LIN {X 0,Y 467.573,Z 511.242,A -85,B 0,C 180,E1 -7527.321,E2 -7527.321} C_VEL
LIN {X 0,Y 467.569,Z 511.24,A -85,B 0,C 180,E1 -7530.665,E2 -7530.665} C_VEL
LIN {X 0,Y 467.618,Z 511.239,A -85,B 0,C 180,E1 -7533.2,E2 -7533.2} C_VEL
LIN {X 0,Y 467.583,Z 511.237,A -85,B 0,C 180,E1 -7536.468,E2 -7536.468} C_VEL
LIN {X 0,Y 467.614,Z 511.233,A -85,B 0,C 180,E1 -7539.777,E2 -7539.777} C_VEL
LIN {X 0,Y 467.599,Z 511.235,A -85,B 0,C 180,E1 -7542.507,E2 -7542.507} C_VEL
LIN {X 0,Y 467.597,Z 511.242,A -85,B 0,C 180,E1 -7545.197,E2 -7545.197} C_VEL
LIN {X 0,Y 467.673,Z 511.225,A -85,B 0,C 180,E1 -7547.855,E2 -7547.855} C_VEL
LIN {X 0,Y 467.673,Z 511.231,A -85,B 0,C 180,E1 -7551.358,E2 -7551.358} C_VEL
LIN {X 0,Y 467.744,Z 511.216,A -85,B 0,C 180,E1 -7553.963,E2 -7553.963} C_VEL
LIN {X 0,Y 467.852,Z 511.208,A -85,B 0,C 180,E1 -7557.417,E2 -7557.417} C_VEL
LIN {X 0,Y 467.873,Z 511.2,A -85,B 0,C 180,E1 -7560,E2 -7560} C_VEL
LIN {X 0,Y 467.858,Z 511.203,A -85,B 0,C 180,E1 -7562.583,E2 -7562.583} C_VEL
LIN {X 0,Y 467.745,Z 511.216,A -85,B 0,C 180,E1 -7566.038,E2 -7566.038} C_VEL
LIN {X 0,Y 467.674,Z 511.226,A -85,B 0,C 180,E1 -7568.643,E2 -7568.643} C_VEL
LIN {X 0,Y 467.648,Z 511.228,A -85,B 0,C 180,E1 -7572.146,E2 -7572.146} C_VEL
LIN {X 0,Y 467.63,Z 511.233,A -85,B 0,C 180,E1 -7575.696,E2 -7575.696} C_VEL
LIN {X 0,Y 467.61,Z 511.235,A -85,B 0,C 180,E1 -7578.765,E2 -7578.765} C_VEL
LIN {X 0,Y 467.573,Z 511.246,A -85,B 0,C 180,E1 -7581.269,E2 -7581.269} C_VEL
LIN {X 0,Y 467.566,Z 511.239,A -85,B 0,C 180,E1 -7583.944,E2 -7583.944} C_VEL
LIN {X 0,Y 467.621,Z 511.233,A -85,B 0,C 180,E1 -7586.8,E2 -7586.8} C_VEL
LIN {X 0,Y 467.583,Z 511.239,A -85,B 0,C 180,E1 -7589.737,E2 -7589.737} C_VEL
LIN {X 0,Y 467.578,Z 511.238,A -85,B 0,C 180,E1 -7592.759,E2 -7592.759} C_VEL
LIN {X 0,Y 467.552,Z 511.241,A -85,B 0,C 180,E1 -7595.89,E2 -7595.89} C_VEL
LIN {X 0,Y 467.578,Z 511.242,A -85,B 0,C 180,E1 -7599.146,E2 -7599.146} C_VEL
LIN {X 0,Y 467.583,Z 511.236,A -85,B 0,C 180,E1 -7602.568,E2 -7602.568} C_VEL
LIN {X 0,Y 467.567,Z 511.242,A -85,B 0,C 180,E1 -7605.054,E2 -7605.054} C_VEL
LIN {X 0,Y 467.622,Z 511.238,A -85,B 0,C 180,E1 -7607.445,E2 -7607.445} C_VEL
LIN {X 0,Y 467.613,Z 511.234,A -85,B 0,C 180,E1 -7610.86,E2 -7610.86} C_VEL
LIN {X 0,Y 467.561,Z 511.239,A -85,B 0,C 180,E1 -7614.261,E2 -7614.261} C_VEL
LIN {X 0,Y 467.582,Z 511.244,A -85,B 0,C 180,E1 -7617.322,E2 -7617.322} C_VEL
LIN {X 0,Y 467.57,Z 511.242,A -85,B 0,C 180,E1 -7620.668,E2 -7620.668} C_VEL
LIN {X 0,Y 467.685,Z 511.313,A -85,B 0,C 180,E1 -7622.784,E2 -7622.784} C_VEL
LIN {X 0,Y 470.344,Z 524.929,A -85,B 0,C 180,E1 -7625.268,E2 -7625.268} C_VEL
LIN {X 0,Y 469.76,Z 538.705,A -85,B 0,C 180,E1 -7627.574,E2 -7627.574} C_VEL
LIN {X 0,Y 468.885,Z 558.208,A -85,B 0,C 180,E1 -7630.786,E2 -7630.786} C_VEL
LIN {X 0,Y 468.378,Z 571.672,A -85,B 0,C 180,E1 -7632.979,E2 -7632.979} C_VEL
LIN {X 0,Y 471.177,Z 592.338,A -85,B 0,C 180,E1 -7633.414,E2 -7633.414} C_VEL
LIN {X 0,Y 470.446,Z 679.842,A -85,B 0,C 180,E1 -7634.79,E2 -7634.79} C_VEL
LIN {X 0,Y 470.108,Z 692.551,A -85,B 0,C 180,E1 -7635.139,E2 -7635.139} C_VEL
LIN {X 0,Y 469.678,Z 705.019,A -85,B 0,C 180,E1 -7635.651,E2 -7635.651} C_VEL
LIN {X 0,Y 469.158,Z 717.567,A -85,B 0,C 180,E1 -7636.354,E2 -7636.354} C_VEL
LIN {X 0,Y 468.644,Z 729.795,A -85,B 0,C 180,E1 -7637.261,E2 -7637.261} C_VEL
LIN {X 0,Y 468.237,Z 739.902,A -85,B 0,C 180,E1 -7638.2,E2 -7638.2} C_VEL
LIN {X 0,Y 467.747,Z 748.542,A -85,B 0,C 180,E1 -7639.175,E2 -7639.175} C_VEL
LIN {X 0,Y 467.406,Z 756.518,A -85,B 0,C 180,E1 -7640.261,E2 -7640.261} C_VEL
LIN {X 0,Y 467.107,Z 764.316,A -85,B 0,C 180,E1 -7641.565,E2 -7641.565} C_VEL
LIN {X 0,Y 466.859,Z 771.486,A -85,B 0,C 180,E1 -7643.083,E2 -7643.083} C_VEL
LIN {X 0,Y 466.781,Z 776.263,A -85,B 0,C 180,E1 -7644.384,E2 -7644.384} C_VEL
LIN {X 0,Y 466.664,Z 779.908,A -85,B 0,C 180,E1 -7645.682,E2 -7645.682} C_VEL
LIN {X 0,Y 466.728,Z 781.794,A -85,B 0,C 180,E1 -7646.547,E2 -7646.547} C_VEL
LIN {X 0,Y 466.701,Z 783.202,A -85,B 0,C 180,E1 -7647.411,E2 -7647.411} C_VEL
LIN {X 0,Y 466.693,Z 784.204,A -85,B 0,C 180,E1 -7648.274,E2 -7648.274} C_VEL
LIN {X 0,Y 466.599,Z 785.018,A -85,B 0,C 180,E1 -7650,E2 -7650} C_VEL
LIN {X 0,Y 466.693,Z 784.171,A -85,B 0,C 180,E1 -7651.726,E2 -7651.726} C_VEL
LIN {X 0,Y 466.701,Z 783.153,A -85,B 0,C 180,E1 -7652.589,E2 -7652.589} C_VEL
LIN {X 0,Y 466.729,Z 781.728,A -85,B 0,C 180,E1 -7653.453,E2 -7653.453} C_VEL
LIN {X 0,Y 466.696,Z 778.735,A -85,B 0,C 180,E1 -7654.751,E2 -7654.751} C_VEL
LIN {X 0,Y 466.765,Z 774.695,A -85,B 0,C 180,E1 -7656.05,E2 -7656.05} C_VEL
LIN {X 0,Y 466.927,Z 768.484,A -85,B 0,C 180,E1 -7657.568,E2 -7657.568} C_VEL
LIN {X 0,Y 467.148,Z 761.707,A -85,B 0,C 180,E1 -7658.871,E2 -7658.871} C_VEL
LIN {X 0,Y 467.479,Z 753.307,A -85,B 0,C 180,E1 -7660.174,E2 -7660.174} C_VEL
LIN {X 0,Y 467.908,Z 744.688,A -85,B 0,C 180,E1 -7661.26,E2 -7661.26} C_VEL
LIN {X 0,Y 468.351,Z 734.541,A -85,B 0,C 180,E1 -7662.301,E2 -7662.301} C_VEL
LIN {X 0,Y 468.939,Z 723.534,A -85,B 0,C 180,E1 -7663.212,E2 -7663.212} C_VEL
LIN {X 0,Y 469.348,Z 711.968,A -85,B 0,C 180,E1 -7663.972,E2 -7663.972} C_VEL
LIN {X 0,Y 469.843,Z 698.703,A -85,B 0,C 180,E1 -7664.62,E2 -7664.62} C_VEL
LIN {X 0,Y 470.25,Z 685.293,A -85,B 0,C 180,E1 -7665.078,E2 -7665.078} C_VEL
LIN {X 0,Y 470.545,Z 671.932,A -85,B 0,C 180,E1 -7665.345,E2 -7665.345} C_VEL
LIN {X 0,Y 471.04,Z 590.105,A -85,B 0,C 180,E1 -7666.624,E2 -7666.624} C_VEL
LIN {X 0,Y 468.329,Z 570.989,A -85,B 0,C 180,E1 -7667.044,E2 -7667.044} C_VEL
LIN {X 0,Y 469.127,Z 550.502,A -85,B 0,C 180,E1 -7670.383,E2 -7670.383} C_VEL
LIN {X 0,Y 469.926,Z 532.596,A -85,B 0,C 180,E1 -7673.348,E2 -7673.348} C_VEL
LIN {X 0,Y 470.213,Z 524.341,A -85,B 0,C 180,E1 -7674.739,E2 -7674.739} C_VEL
LIN {X 0,Y 467.69,Z 511.23,A -85,B 0,C 180,E1 -7677.16,E2 -7677.16} C_VEL
LIN {X 0,Y 467.571,Z 511.246,A -85,B 0,C 180,E1 -7680.733,E2 -7680.733} C_VEL
LIN {X 0,Y 467.586,Z 511.241,A -85,B 0,C 180,E1 -7683.787,E2 -7683.787} C_VEL
LIN {X 0,Y 467.55,Z 511.244,A -85,B 0,C 180,E1 -7687.186,E2 -7687.186} C_VEL
LIN {X 0,Y 467.594,Z 511.239,A -85,B 0,C 180,E1 -7690.262,E2 -7690.262} C_VEL
LIN {X 0,Y 467.617,Z 511.239,A -85,B 0,C 180,E1 -7692.57,E2 -7692.57} C_VEL
LIN {X 0,Y 467.563,Z 511.241,A -85,B 0,C 180,E1 -7696.176,E2 -7696.176} C_VEL
LIN {X 0,Y 467.578,Z 511.244,A -85,B 0,C 180,E1 -7698.722,E2 -7698.722} C_VEL
LIN {X 0,Y 467.562,Z 511.24,A -85,B 0,C 180,E1 -7701.955,E2 -7701.955} C_VEL
LIN {X 0,Y 467.563,Z 511.241,A -85,B 0,C 180,E1 -7705.167,E2 -7705.167} C_VEL
LIN {X 0,Y 467.58,Z 511.239,A -85,B 0,C 180,E1 -7708.259,E2 -7708.259} C_VEL
LIN {X 0,Y 467.577,Z 511.239,A -85,B 0,C 180,E1 -7711.25,E2 -7711.25} C_VEL
LIN {X 0,Y 467.605,Z 511.235,A -85,B 0,C 180,E1 -7714.159,E2 -7714.159} C_VEL
LIN {X 0,Y 467.569,Z 511.245,A -85,B 0,C 180,E1 -7716.995,E2 -7716.995} C_VEL
LIN {X 0,Y 467.616,Z 511.231,A -85,B 0,C 180,E1 -7719.776,E2 -7719.776} C_VEL
LIN {X 0,Y 467.601,Z 511.237,A -85,B 0,C 180,E1 -7722.506,E2 -7722.506} C_VEL
LIN {X 0,Y 467.598,Z 511.238,A -85,B 0,C 180,E1 -7725.196,E2 -7725.196} C_VEL
LIN {X 0,Y 467.648,Z 511.229,A -85,B 0,C 180,E1 -7727.854,E2 -7727.854} C_VEL
LIN {X 0,Y 467.674,Z 511.229,A -85,B 0,C 180,E1 -7731.357,E2 -7731.357} C_VEL
LIN {X 0,Y 467.745,Z 511.214,A -85,B 0,C 180,E1 -7733.962,E2 -7733.962} C_VEL
LIN {X 0,Y 467.851,Z 511.206,A -85,B 0,C 180,E1 -7737.417,E2 -7737.417} C_VEL
LIN {X 0,Y 467.873,Z 511.199,A -85,B 0,C 180,E1 -7740,E2 -7740} C_VEL
LIN {X 0,Y 467.852,Z 511.206,A -85,B 0,C 180,E1 -7742.583,E2 -7742.583} C_VEL
LIN {X 0,Y 467.745,Z 511.216,A -85,B 0,C 180,E1 -7746.037,E2 -7746.037} C_VEL
LIN {X 0,Y 467.673,Z 511.229,A -85,B 0,C 180,E1 -7748.642,E2 -7748.642} C_VEL
LIN {X 0,Y 467.647,Z 511.229,A -85,B 0,C 180,E1 -7752.145,E2 -7752.145} C_VEL
LIN {X 0,Y 467.629,Z 511.233,A -85,B 0,C 180,E1 -7755.695,E2 -7755.695} C_VEL
LIN {X 0,Y 467.608,Z 511.238,A -85,B 0,C 180,E1 -7758.765,E2 -7758.765} C_VEL
LIN {X 0,Y 467.571,Z 511.246,A -85,B 0,C 180,E1 -7761.268,E2 -7761.268} C_VEL
LIN {X 0,Y 467.563,Z 511.244,A -85,B 0,C 180,E1 -7763.943,E2 -7763.943} C_VEL
LIN {X 0,Y 467.618,Z 511.241,A -85,B 0,C 180,E1 -7766.8,E2 -7766.8} C_VEL
LIN {X 0,Y 467.578,Z 511.243,A -85,B 0,C 180,E1 -7769.736,E2 -7769.736} C_VEL
LIN {X 0,Y 467.629,Z 511.278,A -85,B 0,C 180,E1 -7772.383,E2 -7772.383} C_VEL
LIN {X 0,Y 468.698,Z 518.116,A -85,B 0,C 180,E1 -7774.066,E2 -7774.066} C_VEL
LIN {X 0,Y 468.606,Z 522.269,A -85,B 0,C 180,E1 -7775.038,E2 -7775.038} C_VEL
LIN {X 0,Y 471.44,Z 535.638,A -85,B 0,C 180,E1 -7775.384,E2 -7775.384} C_VEL
LIN {X 0,Y 470.589,Z 628.803,A -85,B 0,C 180,E1 -7776.865,E2 -7776.865} C_VEL
LIN {X 0,Y 470.3,Z 642.7,A -85,B 0,C 180,E1 -7777.278,E2 -7777.278} C_VEL
LIN {X 0,Y 470.018,Z 654.766,A -85,B 0,C 180,E1 -7777.81,E2 -7777.81} C_VEL
LIN {X 0,Y 469.536,Z 666.953,A -85,B 0,C 180,E1 -7778.538,E2 -7778.538} C_VEL
LIN {X 0,Y 469.053,Z 678.321,A -85,B 0,C 180,E1 -7779.413,E2 -7779.413} C_VEL
LIN {X 0,Y 468.519,Z 688.987,A -85,B 0,C 180,E1 -7780.448,E2 -7780.448} C_VEL
LIN {X 0,Y 468.053,Z 698.759,A -85,B 0,C 180,E1 -7781.637,E2 -7781.637} C_VEL
LIN {X 0,Y 467.629,Z 706.828,A -85,B 0,C 180,E1 -7782.847,E2 -7782.847} C_VEL
LIN {X 0,Y 467.334,Z 713.616,A -85,B 0,C 180,E1 -7784.105,E2 -7784.105} C_VEL
LIN {X 0,Y 467.068,Z 719.943,A -85,B 0,C 180,E1 -7785.599,E2 -7785.599} C_VEL
LIN {X 0,Y 466.933,Z 723.941,A -85,B 0,C 180,E1 -7786.81,E2 -7786.81} C_VEL
LIN {X 0,Y 466.808,Z 727.024,A -85,B 0,C 180,E1 -7788.02,E2 -7788.02} C_VEL
LIN {X 0,Y 466.633,Z 729.788,A -85,B 0,C 180,E1 -7789.638,E2 -7789.638} C_VEL
LIN {X 0,Y 466.57,Z 730.886,A -85,B 0,C 180,E1 -7790.755,E2 -7790.755} C_VEL
LIN {X 0,Y 466.575,Z 731.291,A -85,B 0,C 180,E1 -7791.861,E2 -7791.861} C_VEL
LIN {X 0,Y 466.571,Z 731.055,A -85,B 0,C 180,E1 -7792.971,E2 -7792.971} C_VEL
LIN {X 0,Y 466.6,Z 729.522,A -85,B 0,C 180,E1 -7794.588,E2 -7794.588} C_VEL
LIN {X 0,Y 466.766,Z 726.76,A -85,B 0,C 180,E1 -7796.145,E2 -7796.145} C_VEL
LIN {X 0,Y 466.914,Z 723.325,A -85,B 0,C 180,E1 -7797.448,E2 -7797.448} C_VEL
LIN {X 0,Y 466.999,Z 720.883,A -85,B 0,C 180,E1 -7798.19,E2 -7798.19} C_VEL
LIN {X 0,Y 466.47,Z 718.546,A -85,B 0,C 180,E1 -7798.854,E2 -7798.854} C_VEL
LIN {X 0,Y 463.785,Z 714.337,A -85,B 0,C 180,E1 -7799.912,E2 -7799.912} C_VEL
LIN {X 0,Y 461.138,Z 709.44,A -85,B 0,C 180,E1 -7800.934,E2 -7800.934} C_VEL
LIN {X 0,Y 460.675,Z 706.022,A -85,B 0,C 180,E1 -7801.532,E2 -7801.532} C_VEL
LIN {X 0,Y 461.128,Z 697.482,A -85,B 0,C 180,E1 -7802.792,E2 -7802.792} C_VEL
LIN {X 0,Y 461.645,Z 688.03,A -85,B 0,C 180,E1 -7803.922,E2 -7803.922} C_VEL
LIN {X 0,Y 462.119,Z 677.677,A -85,B 0,C 180,E1 -7804.918,E2 -7804.918} C_VEL
LIN {X 0,Y 462.601,Z 666.443,A -85,B 0,C 180,E1 -7805.784,E2 -7805.784} C_VEL
LIN {X 0,Y 463.087,Z 653.998,A -85,B 0,C 180,E1 -7806.524,E2 -7806.524} C_VEL
LIN {X 0,Y 463.455,Z 640.905,A -85,B 0,C 180,E1 -7807.088,E2 -7807.088} C_VEL
LIN {X 0,Y 463.693,Z 627.903,A -85,B 0,C 180,E1 -7807.463,E2 -7807.463} C_VEL
LIN {X 0,Y 464.487,Z 535.776,A -85,B 0,C 180,E1 -7808.94,E2 -7808.94} C_VEL
LIN {X 0,Y 461.511,Z 521.937,A -85,B 0,C 180,E1 -7809.294,E2 -7809.294} C_VEL
LIN {X 0,Y 461.424,Z 517.113,A -85,B 0,C 180,E1 -7810.423,E2 -7810.423} C_VEL
LIN {X 0,Y 460.618,Z 512.11,A -85,B 0,C 180,E1 -7811.658,E2 -7811.658} C_VEL
LIN {X 0,Y 460.562,Z 512.118,A -85,B 0,C 180,E1 -7814.965,E2 -7814.965} C_VEL
LIN {X 0,Y 460.608,Z 512.109,A -85,B 0,C 180,E1 -7818.559,E2 -7818.559} C_VEL
LIN {X 0,Y 460.692,Z 512.095,A -85,B 0,C 180,E1 -7822.109,E2 -7822.109} C_VEL
LIN {X 0,Y 460.692,Z 512.101,A -85,B 0,C 180,E1 -7824.748,E2 -7824.748} C_VEL
LIN {X 0,Y 460.823,Z 512.08,A -85,B 0,C 180,E1 -7827.378,E2 -7827.378} C_VEL
LIN {X 0,Y 460.851,Z 512.075,A -85,B 0,C 180,E1 -7830,E2 -7830} C_VEL
LIN {X 0,Y 460.822,Z 512.082,A -85,B 0,C 180,E1 -7832.622,E2 -7832.622} C_VEL
LIN {X 0,Y 460.709,Z 512.093,A -85,B 0,C 180,E1 -7836.13,E2 -7836.13} C_VEL
LIN {X 0,Y 460.626,Z 512.109,A -85,B 0,C 180,E1 -7838.776,E2 -7838.776} C_VEL
LIN {X 0,Y 460.61,Z 512.107,A -85,B 0,C 180,E1 -7842.445,E2 -7842.445} C_VEL
LIN {X 0,Y 460.596,Z 512.106,A -85,B 0,C 180,E1 -7845.997,E2 -7845.997} C_VEL
LIN {X 0,Y 460.567,Z 512.117,A -85,B 0,C 180,E1 -7848.902,E2 -7848.902} C_VEL
LIN {X 0,Y 460.512,Z 512.119,A -85,B 0,C 180,E1 -7851.485,E2 -7851.485} C_VEL
LIN {X 0,Y 460.538,Z 512.114,A -85,B 0,C 180,E1 -7854.332,E2 -7854.332} C_VEL
LIN {X 0,Y 460.575,Z 512.114,A -85,B 0,C 180,E1 -7857.243,E2 -7857.243} C_VEL
LIN {X 0,Y 460.526,Z 512.115,A -85,B 0,C 180,E1 -7860.238,E2 -7860.238} C_VEL
LIN {X 0,Y 460.523,Z 512.12,A -85,B 0,C 180,E1 -7863.324,E2 -7863.324} C_VEL
LIN {X 0,Y 460.474,Z 512.124,A -85,B 0,C 180,E1 -7866.529,E2 -7866.529} C_VEL
LIN {X 0,Y 460.572,Z 512.109,A -85,B 0,C 180,E1 -7869.857,E2 -7869.857} C_VEL
LIN {X 0,Y 460.536,Z 512.12,A -85,B 0,C 180,E1 -7872.904,E2 -7872.904} C_VEL
LIN {X 0,Y 460.516,Z 512.117,A -85,B 0,C 180,E1 -7875.828,E2 -7875.828} C_VEL
LIN {X 0,Y 460.535,Z 512.121,A -85,B 0,C 180,E1 -7878.99,E2 -7878.99} C_VEL
LIN {X 0,Y 460.539,Z 512.119,A -85,B 0,C 180,E1 -7881.269,E2 -7881.269} C_VEL
LIN {X 0,Y 460.505,Z 512.119,A -85,B 0,C 180,E1 -7884.555,E2 -7884.555} C_VEL
LIN {X 0,Y 460.523,Z 512.117,A -85,B 0,C 180,E1 -7887.716,E2 -7887.716} C_VEL
LIN {X 0,Y 460.538,Z 512.117,A -85,B 0,C 180,E1 -7890.769,E2 -7890.769} C_VEL
LIN {X 0,Y 460.559,Z 512.112,A -85,B 0,C 180,E1 -7893.735,E2 -7893.735} C_VEL
LIN {X 0,Y 460.536,Z 512.116,A -85,B 0,C 180,E1 -7896.624,E2 -7896.624} C_VEL
LIN {X 0,Y 460.542,Z 512.117,A -85,B 0,C 180,E1 -7899.453,E2 -7899.453} C_VEL
LIN {X 0,Y 460.549,Z 512.112,A -85,B 0,C 180,E1 -7902.23,E2 -7902.23} C_VEL
LIN {X 0,Y 460.555,Z 512.117,A -85,B 0,C 180,E1 -7904.965,E2 -7904.965} C_VEL
LIN {X 0,Y 460.62,Z 512.105,A -85,B 0,C 180,E1 -7907.667,E2 -7907.667} C_VEL
LIN {X 0,Y 460.62,Z 512.111,A -85,B 0,C 180,E1 -7911.224,E2 -7911.224} C_VEL
LIN {X 0,Y 460.709,Z 512.093,A -85,B 0,C 180,E1 -7913.871,E2 -7913.871} C_VEL
LIN {X 0,Y 460.817,Z 512.085,A -85,B 0,C 180,E1 -7917.378,E2 -7917.378} C_VEL
LIN {X 0,Y 460.844,Z 512.076,A -85,B 0,C 180,E1 -7920,E2 -7920} C_VEL
LIN {X 0,Y 460.824,Z 512.079,A -85,B 0,C 180,E1 -7922.623,E2 -7922.623} C_VEL
LIN {X 0,Y 460.71,Z 512.092,A -85,B 0,C 180,E1 -7926.13,E2 -7926.13} C_VEL
LIN {X 0,Y 460.621,Z 512.106,A -85,B 0,C 180,E1 -7928.777,E2 -7928.777} C_VEL
LIN {X 0,Y 460.604,Z 512.106,A -85,B 0,C 180,E1 -7932.446,E2 -7932.446} C_VEL
LIN {X 0,Y 460.592,Z 512.107,A -85,B 0,C 180,E1 -7935.998,E2 -7935.998} C_VEL
LIN {X 0,Y 460.563,Z 512.114,A -85,B 0,C 180,E1 -7938.903,E2 -7938.903} C_VEL
LIN {X 0,Y 460.508,Z 512.123,A -85,B 0,C 180,E1 -7941.486,E2 -7941.486} C_VEL
LIN {X 0,Y 460.535,Z 512.114,A -85,B 0,C 180,E1 -7944.333,E2 -7944.333} C_VEL
LIN {X 0,Y 460.578,Z 512.116,A -85,B 0,C 180,E1 -7947.244,E2 -7947.244} C_VEL
LIN {X 0,Y 460.525,Z 512.115,A -85,B 0,C 180,E1 -7950.239,E2 -7950.239} C_VEL
LIN {X 0,Y 460.524,Z 512.124,A -85,B 0,C 180,E1 -7953.326,E2 -7953.326} C_VEL
LIN {X 0,Y 460.475,Z 512.122,A -85,B 0,C 180,E1 -7956.53,E2 -7956.53} C_VEL
LIN {X 0,Y 460.554,Z 512.113,A -85,B 0,C 180,E1 -7959.861,E2 -7959.861} C_VEL
LIN {X 0,Y 460.513,Z 512.119,A -85,B 0,C 180,E1 -7962.902,E2 -7962.902} C_VEL
LIN {X 0,Y 460.521,Z 512.118,A -85,B 0,C 180,E1 -7965.83,E2 -7965.83} C_VEL
LIN {X 0,Y 460.541,Z 512.117,A -85,B 0,C 180,E1 -7968.991,E2 -7968.991} C_VEL
LIN {X 0,Y 460.542,Z 512.12,A -85,B 0,C 180,E1 -7971.27,E2 -7971.27} C_VEL
LIN {X 0,Y 460.512,Z 512.117,A -85,B 0,C 180,E1 -7974.555,E2 -7974.555} C_VEL
LIN {X 0,Y 460.532,Z 512.121,A -85,B 0,C 180,E1 -7977.717,E2 -7977.717} C_VEL
LIN {X 0,Y 460.54,Z 512.118,A -85,B 0,C 180,E1 -7980.77,E2 -7980.77} C_VEL
LIN {X 0,Y 460.637,Z 512.174,A -85,B 0,C 180,E1 -7982.554,E2 -7982.554} C_VEL
LIN {X 0,Y 463.311,Z 525.627,A -85,B 0,C 180,E1 -7985.055,E2 -7985.055} C_VEL
LIN {X 0,Y 463.231,Z 531.441,A -85,B 0,C 180,E1 -7986.057,E2 -7986.057} C_VEL
LIN {X 0,Y 462.345,Z 549.328,A -85,B 0,C 180,E1 -7989.071,E2 -7989.071} C_VEL
LIN {X 0,Y 461.463,Z 569.802,A -85,B 0,C 180,E1 -7992.473,E2 -7992.473} C_VEL
LIN {X 0,Y 461.394,Z 571.264,A -85,B 0,C 180,E1 -7992.713,E2 -7992.713} C_VEL
LIN {X 0,Y 464.355,Z 592.628,A -85,B 0,C 180,E1 -7993.179,E2 -7993.179} C_VEL
LIN {X 0,Y 463.544,Z 680.366,A -85,B 0,C 180,E1 -7994.586,E2 -7994.586} C_VEL
LIN {X 0,Y 463.158,Z 693.499,A -85,B 0,C 180,E1 -7994.967,E2 -7994.967} C_VEL
LIN {X 0,Y 462.688,Z 706.737,A -85,B 0,C 180,E1 -7995.542,E2 -7995.542} C_VEL
LIN {X 0,Y 462.156,Z 718.676,A -85,B 0,C 180,E1 -7996.255,E2 -7996.255} C_VEL
LIN {X 0,Y 461.625,Z 730.429,A -85,B 0,C 180,E1 -7997.159,E2 -7997.159} C_VEL
LIN {X 0,Y 461.203,Z 740.514,A -85,B 0,C 180,E1 -7998.129,E2 -7998.129} C_VEL
LIN {X 0,Y 460.633,Z 749.81,A -85,B 0,C 180,E1 -7999.228,E2 -7999.228} C_VEL
LIN {X 0,Y 460.215,Z 758.854,A -85,B 0,C 180,E1 -8000.552,E2 -8000.552} C_VEL
LIN {X 0,Y 459.936,Z 766.143,A -85,B 0,C 180,E1 -8001.875,E2 -8001.875} C_VEL
LIN {X 0,Y 459.747,Z 772.252,A -85,B 0,C 180,E1 -8003.273,E2 -8003.273} C_VEL
LIN {X 0,Y 459.679,Z 777.178,A -85,B 0,C 180,E1 -8004.737,E2 -8004.737} C_VEL
LIN {X 0,Y 459.579,Z 779.494,A -85,B 0,C 180,E1 -8005.615,E2 -8005.615} C_VEL
LIN {X 0,Y 459.626,Z 781.382,A -85,B 0,C 180,E1 -8006.494,E2 -8006.494} C_VEL
LIN {X 0,Y 459.621,Z 782.794,A -85,B 0,C 180,E1 -8007.371,E2 -8007.371} C_VEL
LIN {X 0,Y 459.63,Z 783.797,A -85,B 0,C 180,E1 -8008.248,E2 -8008.248} C_VEL
LIN {X 0,Y 459.531,Z 784.611,A -85,B 0,C 180,E1 -8010,E2 -8010} C_VEL
LIN {X 0,Y 459.63,Z 783.763,A -85,B 0,C 180,E1 -8011.752,E2 -8011.752} C_VEL
LIN {X 0,Y 459.621,Z 782.742,A -85,B 0,C 180,E1 -8012.629,E2 -8012.629} C_VEL
LIN {X 0,Y 459.626,Z 781.315,A -85,B 0,C 180,E1 -8013.506,E2 -8013.506} C_VEL
LIN {X 0,Y 459.627,Z 778.32,A -85,B 0,C 180,E1 -8014.824,E2 -8014.824} C_VEL
LIN {X 0,Y 459.715,Z 773.225,A -85,B 0,C 180,E1 -8016.431,E2 -8016.431} C_VEL
LIN {X 0,Y 459.891,Z 767.031,A -85,B 0,C 180,E1 -8017.905,E2 -8017.905} C_VEL
LIN {X 0,Y 460.181,Z 760.022,A -85,B 0,C 180,E1 -8019.227,E2 -8019.227} C_VEL
LIN {X 0,Y 460.532,Z 751.247,A -85,B 0,C 180,E1 -8020.552,E2 -8020.552} C_VEL
LIN {X 0,Y 461.034,Z 742.268,A -85,B 0,C 180,E1 -8021.653,E2 -8021.653} C_VEL
LIN {X 0,Y 461.56,Z 731.528,A -85,B 0,C 180,E1 -8022.726,E2 -8022.726} C_VEL
LIN {X 0,Y 462.095,Z 720.024,A -85,B 0,C 180,E1 -8023.635,E2 -8023.635} C_VEL
LIN {X 0,Y 462.63,Z 707.504,A -85,B 0,C 180,E1 -8024.404,E2 -8024.404} C_VEL
LIN {X 0,Y 463.15,Z 694.847,A -85,B 0,C 180,E1 -8024.977,E2 -8024.977} C_VEL
LIN {X 0,Y 463.495,Z 682.598,A -85,B 0,C 180,E1 -8025.359,E2 -8025.359} C_VEL
LIN {X 0,Y 463.857,Z 662.673,A -85,B 0,C 180,E1 -8025.713,E2 -8025.713} C_VEL
LIN {X 0,Y 464.27,Z 591.113,A -85,B 0,C 180,E1 -8026.856,E2 -8026.856} C_VEL
LIN {X 0,Y 461.349,Z 570.475,A -85,B 0,C 180,E1 -8027.326,E2 -8027.326} C_VEL
LIN {X 0,Y 462.145,Z 551.497,A -85,B 0,C 180,E1 -8030.473,E2 -8030.473} C_VEL
LIN {X 0,Y 463.065,Z 532.253,A -85,B 0,C 180,E1 -8033.715,E2 -8033.715} C_VEL
LIN {X 0,Y 463.211,Z 525.142,A -85,B 0,C 180,E1 -8034.942,E2 -8034.942} C_VEL
LIN {X 0,Y 460.617,Z 512.11,A -85,B 0,C 180,E1 -8037.406,E2 -8037.406} C_VEL
LIN {X 0,Y 460.511,Z 512.124,A -85,B 0,C 180,E1 -8040.239,E2 -8040.239} C_VEL
LIN {X 0,Y 460.529,Z 512.121,A -85,B 0,C 180,E1 -8043.324,E2 -8043.324} C_VEL
LIN {X 0,Y 460.478,Z 512.13,A -85,B 0,C 180,E1 -8046.528,E2 -8046.528} C_VEL
LIN {X 0,Y 460.574,Z 512.111,A -85,B 0,C 180,E1 -8049.857,E2 -8049.857} C_VEL
LIN {X 0,Y 460.54,Z 512.119,A -85,B 0,C 180,E1 -8052.903,E2 -8052.903} C_VEL
LIN {X 0,Y 460.516,Z 512.117,A -85,B 0,C 180,E1 -8055.828,E2 -8055.828} C_VEL
LIN {X 0,Y 460.53,Z 512.12,A -85,B 0,C 180,E1 -8058.988,E2 -8058.988} C_VEL
LIN {X 0,Y 460.522,Z 512.119,A -85,B 0,C 180,E1 -8061.266,E2 -8061.266} C_VEL
LIN {X 0,Y 460.509,Z 512.123,A -85,B 0,C 180,E1 -8064.554,E2 -8064.554} C_VEL
LIN {X 0,Y 460.527,Z 512.116,A -85,B 0,C 180,E1 -8067.715,E2 -8067.715} C_VEL
LIN {X 0,Y 460.541,Z 512.121,A -85,B 0,C 180,E1 -8070.769,E2 -8070.769} C_VEL
LIN {X 0,Y 460.561,Z 512.112,A -85,B 0,C 180,E1 -8073.734,E2 -8073.734} C_VEL
LIN {X 0,Y 460.539,Z 512.116,A -85,B 0,C 180,E1 -8076.623,E2 -8076.623} C_VEL
LIN {X 0,Y 460.544,Z 512.114,A -85,B 0,C 180,E1 -8079.452,E2 -8079.452} C_VEL
LIN {X 0,Y 460.551,Z 512.113,A -85,B 0,C 180,E1 -8082.229,E2 -8082.229} C_VEL
LIN {X 0,Y 460.557,Z 512.119,A -85,B 0,C 180,E1 -8084.964,E2 -8084.964} C_VEL
LIN {X 0,Y 460.601,Z 512.107,A -85,B 0,C 180,E1 -8087.665,E2 -8087.665} C_VEL
LIN {X 0,Y 460.621,Z 512.109,A -85,B 0,C 180,E1 -8091.223,E2 -8091.223} C_VEL
LIN {X 0,Y 460.709,Z 512.09,A -85,B 0,C 180,E1 -8093.87,E2 -8093.87} C_VEL
LIN {X 0,Y 460.817,Z 512.082,A -85,B 0,C 180,E1 -8097.377,E2 -8097.377} C_VEL
LIN {X 0,Y 460.844,Z 512.075,A -85,B 0,C 180,E1 -8100,E2 -8100} C_VEL
LIN {X 0,Y 460.817,Z 512.083,A -85,B 0,C 180,E1 -8102.622,E2 -8102.622} C_VEL
LIN {X 0,Y 460.709,Z 512.092,A -85,B 0,C 180,E1 -8106.129,E2 -8106.129} C_VEL
LIN {X 0,Y 460.62,Z 512.109,A -85,B 0,C 180,E1 -8108.776,E2 -8108.776} C_VEL
LIN {X 0,Y 460.603,Z 512.108,A -85,B 0,C 180,E1 -8112.445,E2 -8112.445} C_VEL
LIN {X 0,Y 460.59,Z 512.109,A -85,B 0,C 180,E1 -8115.997,E2 -8115.997} C_VEL
LIN {X 0,Y 460.561,Z 512.118,A -85,B 0,C 180,E1 -8118.902,E2 -8118.902} C_VEL
LIN {X 0,Y 460.506,Z 512.124,A -85,B 0,C 180,E1 -8121.486,E2 -8121.486} C_VEL
LIN {X 0,Y 460.533,Z 512.12,A -85,B 0,C 180,E1 -8124.332,E2 -8124.332} C_VEL
LIN {X 0,Y 460.574,Z 512.119,A -85,B 0,C 180,E1 -8127.243,E2 -8127.243} C_VEL
LIN {X 0,Y 460.518,Z 512.121,A -85,B 0,C 180,E1 -8130.239,E2 -8130.239} C_VEL
LIN {X 0,Y 460.613,Z 512.276,A -85,B 0,C 180,E1 -8132.213,E2 -8132.213} C_VEL
LIN {X 0,Y 461.745,Z 519.491,A -85,B 0,C 180,E1 -8134.011,E2 -8134.011} C_VEL
LIN {X 0,Y 461.686,Z 522.905,A -85,B 0,C 180,E1 -8134.793,E2 -8134.793} C_VEL
LIN {X 0,Y 464.681,Z 536.46,A -85,B 0,C 180,E1 -8135.136,E2 -8135.136} C_VEL
LIN {X 0,Y 463.762,Z 629.077,A -85,B 0,C 180,E1 -8136.631,E2 -8136.631} C_VEL
LIN {X 0,Y 463.473,Z 642.341,A -85,B 0,C 180,E1 -8137.025,E2 -8137.025} C_VEL
LIN {X 0,Y 463.188,Z 654.654,A -85,B 0,C 180,E1 -8137.568,E2 -8137.568} C_VEL
LIN {X 0,Y 462.718,Z 666.186,A -85,B 0,C 180,E1 -8138.251,E2 -8138.251} C_VEL
LIN {X 0,Y 462.195,Z 677.921,A -85,B 0,C 180,E1 -8139.152,E2 -8139.152} C_VEL
LIN {X 0,Y 461.723,Z 687.432,A -85,B 0,C 180,E1 -8140.062,E2 -8140.062} C_VEL
LIN {X 0,Y 461.2,Z 696.472,A -85,B 0,C 180,E1 -8141.115,E2 -8141.115} C_VEL
LIN {X 0,Y 460.73,Z 705.187,A -85,B 0,C 180,E1 -8142.37,E2 -8142.37} C_VEL
LIN {X 0,Y 460.376,Z 712.937,A -85,B 0,C 180,E1 -8143.764,E2 -8143.764} C_VEL
LIN {X 0,Y 460.094,Z 718.436,A -85,B 0,C 180,E1 -8144.997,E2 -8144.997} C_VEL
LIN {X 0,Y 459.889,Z 723.865,A -85,B 0,C 180,E1 -8146.554,E2 -8146.554} C_VEL
LIN {X 0,Y 459.783,Z 726.943,A -85,B 0,C 180,E1 -8147.736,E2 -8147.736} C_VEL
LIN {X 0,Y 459.604,Z 729.178,A -85,B 0,C 180,E1 -8148.889,E2 -8148.889} C_VEL
LIN {X 0,Y 459.515,Z 730.708,A -85,B 0,C 180,E1 -8150.033,E2 -8150.033} C_VEL
LIN {X 0,Y 459.482,Z 731.576,A -85,B 0,C 180,E1 -8151.266,E2 -8151.266} C_VEL
LIN {X 0,Y 459.473,Z 731.604,A -85,B 0,C 180,E1 -8152.69,E2 -8152.69} C_VEL
LIN {X 0,Y 459.516,Z 730.548,A -85,B 0,C 180,E1 -8154.154,E2 -8154.154} C_VEL
LIN {X 0,Y 459.622,Z 728.276,A -85,B 0,C 180,E1 -8155.659,E2 -8155.659} C_VEL
LIN {X 0,Y 459.846,Z 724.642,A -85,B 0,C 180,E1 -8157.201,E2 -8157.201} C_VEL
LIN {X 0,Y 460.048,Z 719.338,A -85,B 0,C 180,E1 -8158.813,E2 -8158.813} C_VEL
LIN {X 0,Y 460.308,Z 713.599,A -85,B 0,C 180,E1 -8160.143,E2 -8160.143} C_VEL
LIN {X 0,Y 460.675,Z 706.022,A -85,B 0,C 180,E1 -8161.532,E2 -8161.532} C_VEL
LIN {X 0,Y 460.136,Z 703.69,A -85,B 0,C 180,E1 -8161.927,E2 -8161.927} C_VEL
LIN {X 0,Y 454.869,Z 696.121,A -85,B 0,C 180,E1 -8163.166,E2 -8163.166} C_VEL
LIN {X 0,Y 454.431,Z 693.359,A -85,B 0,C 180,E1 -8163.529,E2 -8163.529} C_VEL
LIN {X 0,Y 454.925,Z 683.4,A -85,B 0,C 180,E1 -8164.616,E2 -8164.616} C_VEL
LIN {X 0,Y 455.496,Z 672.72,A -85,B 0,C 180,E1 -8165.55,E2 -8165.55} C_VEL
LIN {X 0,Y 456.001,Z 660.791,A -85,B 0,C 180,E1 -8166.378,E2 -8166.378} C_VEL
LIN {X 0,Y 456.421,Z 648.899,A -85,B 0,C 180,E1 -8167.001,E2 -8167.001} C_VEL
LIN {X 0,Y 456.739,Z 636.3,A -85,B 0,C 180,E1 -8167.475,E2 -8167.475} C_VEL
LIN {X 0,Y 456.979,Z 623.65,A -85,B 0,C 180,E1 -8167.776,E2 -8167.776} C_VEL
LIN {X 0,Y 457.757,Z 537.021,A -85,B 0,C 180,E1 -8169.175,E2 -8169.175} C_VEL
LIN {X 0,Y 454.588,Z 522.315,A -85,B 0,C 180,E1 -8169.556,E2 -8169.556} C_VEL
LIN {X 0,Y 454.375,Z 517.725,A -85,B 0,C 180,E1 -8170.648,E2 -8170.648} C_VEL
LIN {X 0,Y 453.565,Z 512.989,A -85,B 0,C 180,E1 -8171.83,E2 -8171.83} C_VEL
LIN {X 0,Y 453.537,Z 512.994,A -85,B 0,C 180,E1 -8174.727,E2 -8174.727} C_VEL
LIN {X 0,Y 453.557,Z 512.985,A -85,B 0,C 180,E1 -8178.379,E2 -8178.379} C_VEL
LIN {X 0,Y 453.649,Z 512.972,A -85,B 0,C 180,E1 -8181.985,E2 -8181.985} C_VEL
LIN {X 0,Y 453.665,Z 512.975,A -85,B 0,C 180,E1 -8184.667,E2 -8184.667} C_VEL
LIN {X 0,Y 453.763,Z 512.96,A -85,B 0,C 180,E1 -8187.337,E2 -8187.337} C_VEL
LIN {X 0,Y 453.821,Z 512.95,A -85,B 0,C 180,E1 -8190,E2 -8190} C_VEL
LIN {X 0,Y 453.763,Z 512.962,A -85,B 0,C 180,E1 -8192.663,E2 -8192.663} C_VEL
LIN {X 0,Y 453.676,Z 512.969,A -85,B 0,C 180,E1 -8196.225,E2 -8196.225} C_VEL
LIN {X 0,Y 453.589,Z 512.987,A -85,B 0,C 180,E1 -8198.913,E2 -8198.913} C_VEL
LIN {X 0,Y 453.56,Z 512.986,A -85,B 0,C 180,E1 -8202.529,E2 -8202.529} C_VEL
LIN {X 0,Y 453.541,Z 512.986,A -85,B 0,C 180,E1 -8206.196,E2 -8206.196} C_VEL
LIN {X 0,Y 453.517,Z 512.996,A -85,B 0,C 180,E1 -8209.041,E2 -8209.041} C_VEL
LIN {X 0,Y 453.472,Z 512.994,A -85,B 0,C 180,E1 -8211.836,E2 -8211.836} C_VEL
LIN {X 0,Y 453.51,Z 512.994,A -85,B 0,C 180,E1 -8214.734,E2 -8214.734} C_VEL
LIN {X 0,Y 453.534,Z 512.986,A -85,B 0,C 180,E1 -8217.961,E2 -8217.961} C_VEL
LIN {X 0,Y 453.479,Z 512.998,A -85,B 0,C 180,E1 -8220.758,E2 -8220.758} C_VEL
LIN {X 0,Y 453.472,Z 512.994,A -85,B 0,C 180,E1 -8223.912,E2 -8223.912} C_VEL
LIN {X 0,Y 453.466,Z 513.001,A -85,B 0,C 180,E1 -8227.187,E2 -8227.187} C_VEL
LIN {X 0,Y 453.527,Z 512.99,A -85,B 0,C 180,E1 -8229.445,E2 -8229.445} C_VEL
LIN {X 0,Y 453.485,Z 513,A -85,B 0,C 180,E1 -8232.991,E2 -8232.991} C_VEL
LIN {X 0,Y 453.469,Z 512.995,A -85,B 0,C 180,E1 -8235.78,E2 -8235.78} C_VEL
LIN {X 0,Y 453.488,Z 512.992,A -85,B 0,C 180,E1 -8238.211,E2 -8238.211} C_VEL
LIN {X 0,Y 453.524,Z 512.992,A -85,B 0,C 180,E1 -8240.787,E2 -8240.787} C_VEL
LIN {X 0,Y 453.449,Z 512.997,A -85,B 0,C 180,E1 -8243.917,E2 -8243.917} C_VEL
LIN {X 0,Y 453.474,Z 513.001,A -85,B 0,C 180,E1 -8247.151,E2 -8247.151} C_VEL
LIN {X 0,Y 453.505,Z 512.99,A -85,B 0,C 180,E1 -8250.271,E2 -8250.271} C_VEL
LIN {X 0,Y 453.504,Z 512.996,A -85,B 0,C 180,E1 -8253.294,E2 -8253.294} C_VEL
LIN {X 0,Y 453.494,Z 512.991,A -85,B 0,C 180,E1 -8256.239,E2 -8256.239} C_VEL
LIN {X 0,Y 453.474,Z 513.002,A -85,B 0,C 180,E1 -8259.118,E2 -8259.118} C_VEL
LIN {X 0,Y 453.502,Z 512.99,A -85,B 0,C 180,E1 -8261.945,E2 -8261.945} C_VEL
LIN {X 0,Y 453.53,Z 512.989,A -85,B 0,C 180,E1 -8264.726,E2 -8264.726} C_VEL
LIN {X 0,Y 453.592,Z 512.983,A -85,B 0,C 180,E1 -8267.472,E2 -8267.472} C_VEL
LIN {X 0,Y 453.584,Z 512.987,A -85,B 0,C 180,E1 -8271.087,E2 -8271.087} C_VEL
LIN {X 0,Y 453.675,Z 512.97,A -85,B 0,C 180,E1 -8273.775,E2 -8273.775} C_VEL
LIN {X 0,Y 453.758,Z 512.965,A -85,B 0,C 180,E1 -8277.337,E2 -8277.337} C_VEL
LIN {X 0,Y 453.814,Z 512.951,A -85,B 0,C 180,E1 -8280,E2 -8280} C_VEL
LIN {X 0,Y 453.765,Z 512.959,A -85,B 0,C 180,E1 -8282.664,E2 -8282.664} C_VEL
LIN {X 0,Y 453.676,Z 512.968,A -85,B 0,C 180,E1 -8286.226,E2 -8286.226} C_VEL
LIN {X 0,Y 453.585,Z 512.984,A -85,B 0,C 180,E1 -8288.914,E2 -8288.914} C_VEL
LIN {X 0,Y 453.555,Z 512.984,A -85,B 0,C 180,E1 -8292.53,E2 -8292.53} C_VEL
LIN {X 0,Y 453.537,Z 512.986,A -85,B 0,C 180,E1 -8296.197,E2 -8296.197} C_VEL
LIN {X 0,Y 453.513,Z 512.994,A -85,B 0,C 180,E1 -8299.042,E2 -8299.042} C_VEL
LIN {X 0,Y 453.469,Z 512.996,A -85,B 0,C 180,E1 -8301.837,E2 -8301.837} C_VEL
LIN {X 0,Y 453.507,Z 512.991,A -85,B 0,C 180,E1 -8304.735,E2 -8304.735} C_VEL
LIN {X 0,Y 453.532,Z 512.987,A -85,B 0,C 180,E1 -8307.962,E2 -8307.962} C_VEL
LIN {X 0,Y 453.479,Z 512.995,A -85,B 0,C 180,E1 -8310.76,E2 -8310.76} C_VEL
LIN {X 0,Y 453.473,Z 512.995,A -85,B 0,C 180,E1 -8313.914,E2 -8313.914} C_VEL
LIN {X 0,Y 453.466,Z 513.001,A -85,B 0,C 180,E1 -8317.189,E2 -8317.189} C_VEL
LIN {X 0,Y 453.513,Z 512.995,A -85,B 0,C 180,E1 -8319.448,E2 -8319.448} C_VEL
LIN {X 0,Y 453.465,Z 512.998,A -85,B 0,C 180,E1 -8322.995,E2 -8322.995} C_VEL
LIN {X 0,Y 453.474,Z 512.996,A -85,B 0,C 180,E1 -8325.781,E2 -8325.781} C_VEL
LIN {X 0,Y 453.494,Z 512.991,A -85,B 0,C 180,E1 -8328.212,E2 -8328.212} C_VEL
LIN {X 0,Y 453.529,Z 512.988,A -85,B 0,C 180,E1 -8330.789,E2 -8330.789} C_VEL
LIN {X 0,Y 453.455,Z 512.998,A -85,B 0,C 180,E1 -8333.918,E2 -8333.918} C_VEL
LIN {X 0,Y 453.483,Z 513,A -85,B 0,C 180,E1 -8337.152,E2 -8337.152} C_VEL
LIN {X 0,Y 453.476,Z 512.998,A -85,B 0,C 180,E1 -8340.269,E2 -8340.269} C_VEL
LIN {X 0,Y 453.575,Z 513.106,A -85,B 0,C 180,E1 -8342.332,E2 -8342.332} C_VEL
LIN {X 0,Y 456.344,Z 526.822,A -85,B 0,C 180,E1 -8344.928,E2 -8344.928} C_VEL
LIN {X 0,Y 456.422,Z 531.055,A -85,B 0,C 180,E1 -8345.677,E2 -8345.677} C_VEL
LIN {X 0,Y 455.381,Z 550.305,A -85,B 0,C 180,E1 -8348.973,E2 -8348.973} C_VEL
LIN {X 0,Y 454.435,Z 570.899,A -85,B 0,C 180,E1 -8352.448,E2 -8352.448} C_VEL
LIN {X 0,Y 457.537,Z 593.117,A -85,B 0,C 180,E1 -8352.94,E2 -8352.94} C_VEL
LIN {X 0,Y 456.711,Z 679.701,A -85,B 0,C 180,E1 -8354.349,E2 -8354.349} C_VEL
LIN {X 0,Y 456.325,Z 692.926,A -85,B 0,C 180,E1 -8354.736,E2 -8354.736} C_VEL
LIN {X 0,Y 455.811,Z 706.215,A -85,B 0,C 180,E1 -8355.319,E2 -8355.319} C_VEL
LIN {X 0,Y 455.206,Z 718.183,A -85,B 0,C 180,E1 -8356.041,E2 -8356.041} C_VEL
LIN {X 0,Y 454.637,Z 729.953,A -85,B 0,C 180,E1 -8356.958,E2 -8356.958} C_VEL
LIN {X 0,Y 454.211,Z 740.055,A -85,B 0,C 180,E1 -8357.943,E2 -8357.943} C_VEL
LIN {X 0,Y 453.629,Z 749.365,A -85,B 0,C 180,E1 -8359.06,E2 -8359.06} C_VEL
LIN {X 0,Y 453.178,Z 758.418,A -85,B 0,C 180,E1 -8360.403,E2 -8360.403} C_VEL
LIN {X 0,Y 452.865,Z 765.713,A -85,B 0,C 180,E1 -8361.747,E2 -8361.747} C_VEL
LIN {X 0,Y 452.696,Z 770.639,A -85,B 0,C 180,E1 -8362.866,E2 -8362.866} C_VEL
LIN {X 0,Y 452.576,Z 775.425,A -85,B 0,C 180,E1 -8364.207,E2 -8364.207} C_VEL
LIN {X 0,Y 452.5,Z 779.081,A -85,B 0,C 180,E1 -8365.546,E2 -8365.546} C_VEL
LIN {X 0,Y 452.525,Z 780.969,A -85,B 0,C 180,E1 -8366.438,E2 -8366.438} C_VEL
LIN {X 0,Y 452.543,Z 782.385,A -85,B 0,C 180,E1 -8367.33,E2 -8367.33} C_VEL
LIN {X 0,Y 452.538,Z 783.388,A -85,B 0,C 180,E1 -8368.22,E2 -8368.22} C_VEL
LIN {X 0,Y 452.49,Z 783.994,A -85,B 0,C 180,E1 -8369.11,E2 -8369.11} C_VEL
LIN {X 0,Y 452.464,Z 784.204,A -85,B 0,C 180,E1 -8370,E2 -8370} C_VEL
LIN {X 0,Y 452.49,Z 783.978,A -85,B 0,C 180,E1 -8370.89,E2 -8370.89} C_VEL
LIN {X 0,Y 452.538,Z 783.354,A -85,B 0,C 180,E1 -8371.78,E2 -8371.78} C_VEL
LIN {X 0,Y 452.543,Z 782.332,A -85,B 0,C 180,E1 -8372.67,E2 -8372.67} C_VEL
LIN {X 0,Y 452.525,Z 780.901,A -85,B 0,C 180,E1 -8373.562,E2 -8373.562} C_VEL
LIN {X 0,Y 452.558,Z 777.904,A -85,B 0,C 180,E1 -8374.9,E2 -8374.9} C_VEL
LIN {X 0,Y 452.611,Z 773.303,A -85,B 0,C 180,E1 -8376.396,E2 -8376.396} C_VEL
LIN {X 0,Y 452.78,Z 767.63,A -85,B 0,C 180,E1 -8377.806,E2 -8377.806} C_VEL
LIN {X 0,Y 453.064,Z 760.841,A -85,B 0,C 180,E1 -8379.149,E2 -8379.149} C_VEL
LIN {X 0,Y 453.439,Z 752.429,A -85,B 0,C 180,E1 -8380.493,E2 -8380.493} C_VEL
LIN {X 0,Y 453.939,Z 743.805,A -85,B 0,C 180,E1 -8381.611,E2 -8381.611} C_VEL
LIN {X 0,Y 454.417,Z 734.143,A -85,B 0,C 180,E1 -8382.638,E2 -8382.638} C_VEL
LIN {X 0,Y 455.053,Z 722.646,A -85,B 0,C 180,E1 -8383.622,E2 -8383.622} C_VEL
LIN {X 0,Y 455.522,Z 711.084,A -85,B 0,C 180,E1 -8384.405,E2 -8384.405} C_VEL
LIN {X 0,Y 456.057,Z 699.136,A -85,B 0,C 180,E1 -8385.016,E2 -8385.016} C_VEL
LIN {X 0,Y 456.517,Z 685.373,A -85,B 0,C 180,E1 -8385.514,E2 -8385.514} C_VEL
LIN {X 0,Y 456.845,Z 672.938,A -85,B 0,C 180,E1 -8385.789,E2 -8385.789} C_VEL
LIN {X 0,Y 457.46,Z 591.684,A -85,B 0,C 180,E1 -8387.104,E2 -8387.104} C_VEL
LIN {X 0,Y 454.392,Z 570.081,A -85,B 0,C 180,E1 -8387.601,E2 -8387.601} C_VEL
LIN {X 0,Y 455.214,Z 551.13,A -85,B 0,C 180,E1 -8390.799,E2 -8390.799} C_VEL
LIN {X 0,Y 456.231,Z 531.93,A -85,B 0,C 180,E1 -8394.092,E2 -8394.092} C_VEL
LIN {X 0,Y 456.273,Z 526.438,A -85,B 0,C 180,E1 -8395.06,E2 -8395.06} C_VEL
LIN {X 0,Y 453.559,Z 512.988,A -85,B 0,C 180,E1 -8397.638,E2 -8397.638} C_VEL
LIN {X 0,Y 453.477,Z 513.002,A -85,B 0,C 180,E1 -8400.759,E2 -8400.759} C_VEL
LIN {X 0,Y 453.478,Z 513,A -85,B 0,C 180,E1 -8403.912,E2 -8403.912} C_VEL
LIN {X 0,Y 453.47,Z 512.999,A -85,B 0,C 180,E1 -8407.187,E2 -8407.187} C_VEL
LIN {X 0,Y 453.529,Z 512.989,A -85,B 0,C 180,E1 -8409.444,E2 -8409.444} C_VEL
LIN {X 0,Y 453.49,Z 512.997,A -85,B 0,C 180,E1 -8412.991,E2 -8412.991} C_VEL
LIN {X 0,Y 453.47,Z 512.995,A -85,B 0,C 180,E1 -8415.779,E2 -8415.779} C_VEL
LIN {X 0,Y 453.478,Z 512.994,A -85,B 0,C 180,E1 -8418.209,E2 -8418.209} C_VEL
LIN {X 0,Y 453.506,Z 512.995,A -85,B 0,C 180,E1 -8420.79,E2 -8420.79} C_VEL
LIN {X 0,Y 453.453,Z 512.997,A -85,B 0,C 180,E1 -8423.917,E2 -8423.917} C_VEL
LIN {X 0,Y 453.478,Z 512.998,A -85,B 0,C 180,E1 -8427.15,E2 -8427.15} C_VEL
LIN {X 0,Y 453.508,Z 512.991,A -85,B 0,C 180,E1 -8430.27,E2 -8430.27} C_VEL
LIN {X 0,Y 453.507,Z 512.993,A -85,B 0,C 180,E1 -8433.294,E2 -8433.294} C_VEL
LIN {X 0,Y 453.496,Z 512.989,A -85,B 0,C 180,E1 -8436.238,E2 -8436.238} C_VEL
LIN {X 0,Y 453.475,Z 512.996,A -85,B 0,C 180,E1 -8439.117,E2 -8439.117} C_VEL
LIN {X 0,Y 453.504,Z 512.99,A -85,B 0,C 180,E1 -8441.944,E2 -8441.944} C_VEL
LIN {X 0,Y 453.532,Z 512.992,A -85,B 0,C 180,E1 -8444.726,E2 -8444.726} C_VEL
LIN {X 0,Y 453.555,Z 512.986,A -85,B 0,C 180,E1 -8447.47,E2 -8447.47} C_VEL
LIN {X 0,Y 453.584,Z 512.986,A -85,B 0,C 180,E1 -8451.086,E2 -8451.086} C_VEL
LIN {X 0,Y 453.675,Z 512.967,A -85,B 0,C 180,E1 -8453.774,E2 -8453.774} C_VEL
LIN {X 0,Y 453.757,Z 512.962,A -85,B 0,C 180,E1 -8457.336,E2 -8457.336} C_VEL
LIN {X 0,Y 453.814,Z 512.951,A -85,B 0,C 180,E1 -8460,E2 -8460} C_VEL
LIN {X 0,Y 453.758,Z 512.963,A -85,B 0,C 180,E1 -8462.663,E2 -8462.663} C_VEL
LIN {X 0,Y 453.675,Z 512.969,A -85,B 0,C 180,E1 -8466.225,E2 -8466.225} C_VEL
LIN {X 0,Y 453.584,Z 512.986,A -85,B 0,C 180,E1 -8468.913,E2 -8468.913} C_VEL
LIN {X 0,Y 453.553,Z 512.987,A -85,B 0,C 180,E1 -8472.529,E2 -8472.529} C_VEL
LIN {X 0,Y 453.535,Z 512.988,A -85,B 0,C 180,E1 -8476.196,E2 -8476.196} C_VEL
LIN {X 0,Y 453.511,Z 512.996,A -85,B 0,C 180,E1 -8479.041,E2 -8479.041} C_VEL
LIN {X 0,Y 453.467,Z 512.999,A -85,B 0,C 180,E1 -8481.836,E2 -8481.836} C_VEL
LIN {X 0,Y 453.504,Z 512.998,A -85,B 0,C 180,E1 -8484.734,E2 -8484.734} C_VEL
LIN {X 0,Y 453.529,Z 512.993,A -85,B 0,C 180,E1 -8487.961,E2 -8487.961} C_VEL
LIN {X 0,Y 453.526,Z 512.995,A -85,B 0,C 180,E1 -8491.54,E2 -8491.54} C_VEL
LIN {X 0,Y 453.558,Z 513.146,A -85,B 0,C 180,E1 -8491.988,E2 -8491.988} C_VEL
LIN {X 0,Y 454.769,Z 520.286,A -85,B 0,C 180,E1 -8493.803,E2 -8493.803} C_VEL
LIN {X 0,Y 454.753,Z 523.201,A -85,B 0,C 180,E1 -8494.506,E2 -8494.506} C_VEL
LIN {X 0,Y 457.909,Z 537.432,A -85,B 0,C 180,E1 -8494.882,E2 -8494.882} C_VEL
LIN {X 0,Y 456.945,Z 629.549,A -85,B 0,C 180,E1 -8496.394,E2 -8496.394} C_VEL
LIN {X 0,Y 456.62,Z 643.386,A -85,B 0,C 180,E1 -8496.815,E2 -8496.815} C_VEL
LIN {X 0,Y 456.276,Z 656.246,A -85,B 0,C 180,E1 -8497.405,E2 -8497.405} C_VEL
LIN {X 0,Y 455.78,Z 668.219,A -85,B 0,C 180,E1 -8498.151,E2 -8498.151} C_VEL
LIN {X 0,Y 455.282,Z 678.655,A -85,B 0,C 180,E1 -8498.978,E2 -8498.978} C_VEL
LIN {X 0,Y 454.781,Z 688.342,A -85,B 0,C 180,E1 -8499.927,E2 -8499.927} C_VEL
LIN {X 0,Y 454.197,Z 697.716,A -85,B 0,C 180,E1 -8501.052,E2 -8501.052} C_VEL
LIN {X 0,Y 453.656,Z 707.017,A -85,B 0,C 180,E1 -8502.452,E2 -8502.452} C_VEL
LIN {X 0,Y 453.314,Z 714.128,A -85,B 0,C 180,E1 -8503.79,E2 -8503.79} C_VEL
LIN {X 0,Y 453.035,Z 719.5,A -85,B 0,C 180,E1 -8505.047,E2 -8505.047} C_VEL
LIN {X 0,Y 452.832,Z 723.81,A -85,B 0,C 180,E1 -8506.312,E2 -8506.312} C_VEL
LIN {X 0,Y 452.728,Z 727.02,A -85,B 0,C 180,E1 -8507.525,E2 -8507.525} C_VEL
LIN {X 0,Y 452.487,Z 730.269,A -85,B 0,C 180,E1 -8509.283,E2 -8509.283} C_VEL
LIN {X 0,Y 452.403,Z 731.835,A -85,B 0,C 180,E1 -8510.962,E2 -8510.962} C_VEL
LIN {X 0,Y 452.409,Z 732.007,A -85,B 0,C 180,E1 -8512.711,E2 -8512.711} C_VEL
LIN {X 0,Y 452.429,Z 731.238,A -85,B 0,C 180,E1 -8513.877,E2 -8513.877} C_VEL
LIN {X 0,Y 452.505,Z 729.23,A -85,B 0,C 180,E1 -8515.401,E2 -8515.401} C_VEL
LIN {X 0,Y 452.759,Z 725.554,A -85,B 0,C 180,E1 -8517.093,E2 -8517.093} C_VEL
LIN {X 0,Y 452.934,Z 720.928,A -85,B 0,C 180,E1 -8518.584,E2 -8518.584} C_VEL
LIN {X 0,Y 453.216,Z 715.223,A -85,B 0,C 180,E1 -8519.994,E2 -8519.994} C_VEL
LIN {X 0,Y 453.571,Z 708.638,A -85,B 0,C 180,E1 -8521.293,E2 -8521.293} C_VEL
LIN {X 0,Y 454.01,Z 700.578,A -85,B 0,C 180,E1 -8522.58,E2 -8522.58} C_VEL
LIN {X 0,Y 454.431,Z 693.359,A -85,B 0,C 180,E1 -8523.529,E2 -8523.529} C_VEL
LIN {X 0,Y 454.157,Z 689.135,A -85,B 0,C 180,E1 -8524.047,E2 -8524.047} C_VEL
LIN {X 0,Y 451.817,Z 682.047,A -85,B 0,C 180,E1 -8524.87,E2 -8524.87} C_VEL
LIN {X 0,Y 449.297,Z 674.484,A -85,B 0,C 180,E1 -8525.624,E2 -8525.624} C_VEL
LIN {X 0,Y 448.744,Z 669.508,A -85,B 0,C 180,E1 -8526.027,E2 -8526.027} C_VEL
LIN {X 0,Y 449.26,Z 657.627,A -85,B 0,C 180,E1 -8526.796,E2 -8526.796} C_VEL
LIN {X 0,Y 449.649,Z 645.561,A -85,B 0,C 180,E1 -8527.386,E2 -8527.386} C_VEL
LIN {X 0,Y 449.946,Z 633.237,A -85,B 0,C 180,E1 -8527.807,E2 -8527.807} C_VEL
LIN {X 0,Y 450.185,Z 617.652,A -85,B 0,C 180,E1 -8528.117,E2 -8528.117} C_VEL
LIN {X 0,Y 450.903,Z 537.866,A -85,B 0,C 180,E1 -8529.428,E2 -8529.428} C_VEL
LIN {X 0,Y 447.626,Z 522.589,A -85,B 0,C 180,E1 -8529.846,E2 -8529.846} C_VEL
LIN {X 0,Y 447.084,Z 517.067,A -85,B 0,C 180,E1 -8531.201,E2 -8531.201} C_VEL
LIN {X 0,Y 446.488,Z 513.871,A -85,B 0,C 180,E1 -8532.007,E2 -8532.007} C_VEL
LIN {X 0,Y 446.504,Z 513.867,A -85,B 0,C 180,E1 -8534.48,E2 -8534.48} C_VEL
LIN {X 0,Y 446.514,Z 513.861,A -85,B 0,C 180,E1 -8538.193,E2 -8538.193} C_VEL
LIN {X 0,Y 446.597,Z 513.85,A -85,B 0,C 180,E1 -8541.858,E2 -8541.858} C_VEL
LIN {X 0,Y 446.64,Z 513.849,A -85,B 0,C 180,E1 -8544.583,E2 -8544.583} C_VEL
LIN {X 0,Y 446.707,Z 513.84,A -85,B 0,C 180,E1 -8547.295,E2 -8547.295} C_VEL
LIN {X 0,Y 446.791,Z 513.826,A -85,B 0,C 180,E1 -8550,E2 -8550} C_VEL
LIN {X 0,Y 446.706,Z 513.842,A -85,B 0,C 180,E1 -8552.705,E2 -8552.705} C_VEL
LIN {X 0,Y 446.645,Z 513.845,A -85,B 0,C 180,E1 -8556.324,E2 -8556.324} C_VEL
LIN {X 0,Y 446.535,Z 513.865,A -85,B 0,C 180,E1 -8559.055,E2 -8559.055} C_VEL
LIN {X 0,Y 446.518,Z 513.865,A -85,B 0,C 180,E1 -8562.729,E2 -8562.729} C_VEL
LIN {X 0,Y 446.492,Z 513.864,A -85,B 0,C 180,E1 -8566.228,E2 -8566.228} C_VEL
LIN {X 0,Y 446.466,Z 513.87,A -85,B 0,C 180,E1 -8569.303,E2 -8569.303} C_VEL
LIN {X 0,Y 446.414,Z 513.873,A -85,B 0,C 180,E1 -8572.199,E2 -8572.199} C_VEL
LIN {X 0,Y 446.453,Z 513.874,A -85,B 0,C 180,E1 -8575.152,E2 -8575.152} C_VEL
LIN {X 0,Y 446.479,Z 513.865,A -85,B 0,C 180,E1 -8578.178,E2 -8578.178} C_VEL
LIN {X 0,Y 446.428,Z 513.876,A -85,B 0,C 180,E1 -8581.299,E2 -8581.299} C_VEL
LIN {X 0,Y 446.424,Z 513.874,A -85,B 0,C 180,E1 -8584.522,E2 -8584.522} C_VEL
LIN {X 0,Y 446.433,Z 513.871,A -85,B 0,C 180,E1 -8588.083,E2 -8588.083} C_VEL
LIN {X 0,Y 446.441,Z 513.876,A -85,B 0,C 180,E1 -8590.92,E2 -8590.92} C_VEL
LIN {X 0,Y 446.438,Z 513.87,A -85,B 0,C 180,E1 -8593.84,E2 -8593.84} C_VEL
LIN {X 0,Y 446.439,Z 513.871,A -85,B 0,C 180,E1 -8596.397,E2 -8596.397} C_VEL
LIN {X 0,Y 446.461,Z 513.868,A -85,B 0,C 180,E1 -8599.805,E2 -8599.805} C_VEL
LIN {X 0,Y 446.426,Z 513.871,A -85,B 0,C 180,E1 -8602.124,E2 -8602.124} C_VEL
LIN {X 0,Y 446.422,Z 513.875,A -85,B 0,C 180,E1 -8605.477,E2 -8605.477} C_VEL
LIN {X 0,Y 446.41,Z 513.876,A -85,B 0,C 180,E1 -8608.7,E2 -8608.7} C_VEL
LIN {X 0,Y 446.475,Z 513.866,A -85,B 0,C 180,E1 -8611.821,E2 -8611.821} C_VEL
LIN {X 0,Y 446.449,Z 513.873,A -85,B 0,C 180,E1 -8614.848,E2 -8614.848} C_VEL
LIN {X 0,Y 446.438,Z 513.87,A -85,B 0,C 180,E1 -8618.245,E2 -8618.245} C_VEL
LIN {X 0,Y 446.447,Z 513.871,A -85,B 0,C 180,E1 -8621.649,E2 -8621.649} C_VEL
LIN {X 0,Y 446.498,Z 513.863,A -85,B 0,C 180,E1 -8624.48,E2 -8624.48} C_VEL
LIN {X 0,Y 446.531,Z 513.858,A -85,B 0,C 180,E1 -8628.194,E2 -8628.194} C_VEL
LIN {X 0,Y 446.591,Z 513.852,A -85,B 0,C 180,E1 -8631.858,E2 -8631.858} C_VEL
LIN {X 0,Y 446.644,Z 513.846,A -85,B 0,C 180,E1 -8634.583,E2 -8634.583} C_VEL
LIN {X 0,Y 446.702,Z 513.844,A -85,B 0,C 180,E1 -8637.295,E2 -8637.295} C_VEL
LIN {X 0,Y 446.785,Z 513.827,A -85,B 0,C 180,E1 -8640,E2 -8640} C_VEL
LIN {X 0,Y 446.709,Z 513.838,A -85,B 0,C 180,E1 -8642.706,E2 -8642.706} C_VEL
LIN {X 0,Y 446.644,Z 513.844,A -85,B 0,C 180,E1 -8646.324,E2 -8646.324} C_VEL
LIN {X 0,Y 446.531,Z 513.864,A -85,B 0,C 180,E1 -8649.056,E2 -8649.056} C_VEL
LIN {X 0,Y 446.515,Z 513.862,A -85,B 0,C 180,E1 -8652.73,E2 -8652.73} C_VEL
LIN {X 0,Y 446.488,Z 513.864,A -85,B 0,C 180,E1 -8656.229,E2 -8656.229} C_VEL
LIN {X 0,Y 446.462,Z 513.875,A -85,B 0,C 180,E1 -8659.304,E2 -8659.304} C_VEL
LIN {X 0,Y 446.411,Z 513.873,A -85,B 0,C 180,E1 -8662.2,E2 -8662.2} C_VEL
LIN {X 0,Y 446.452,Z 513.875,A -85,B 0,C 180,E1 -8665.153,E2 -8665.153} C_VEL
LIN {X 0,Y 446.478,Z 513.865,A -85,B 0,C 180,E1 -8668.18,E2 -8668.18} C_VEL
LIN {X 0,Y 446.428,Z 513.88,A -85,B 0,C 180,E1 -8671.3,E2 -8671.3} C_VEL
LIN {X 0,Y 446.425,Z 513.872,A -85,B 0,C 180,E1 -8674.524,E2 -8674.524} C_VEL
LIN {X 0,Y 446.426,Z 513.872,A -85,B 0,C 180,E1 -8678.083,E2 -8678.083} C_VEL
LIN {X 0,Y 446.424,Z 513.875,A -85,B 0,C 180,E1 -8680.919,E2 -8680.919} C_VEL
LIN {X 0,Y 446.42,Z 513.874,A -85,B 0,C 180,E1 -8683.844,E2 -8683.844} C_VEL
LIN {X 0,Y 446.444,Z 513.869,A -85,B 0,C 180,E1 -8686.398,E2 -8686.398} C_VEL
LIN {X 0,Y 446.467,Z 513.869,A -85,B 0,C 180,E1 -8689.806,E2 -8689.806} C_VEL
LIN {X 0,Y 446.431,Z 513.871,A -85,B 0,C 180,E1 -8692.125,E2 -8692.125} C_VEL
LIN {X 0,Y 446.43,Z 513.879,A -85,B 0,C 180,E1 -8695.478,E2 -8695.478} C_VEL
LIN {X 0,Y 446.417,Z 513.877,A -85,B 0,C 180,E1 -8698.701,E2 -8698.701} C_VEL
LIN {X 0,Y 446.505,Z 513.908,A -85,B 0,C 180,E1 -8702.079,E2 -8702.079} C_VEL
LIN {X 0,Y 449.084,Z 526.493,A -85,B 0,C 180,E1 -8704.51,E2 -8704.51} C_VEL
LIN {X 0,Y 449.57,Z 530.22,A -85,B 0,C 180,E1 -8705.202,E2 -8705.202} C_VEL
LIN {X 0,Y 448.531,Z 548.52,A -85,B 0,C 180,E1 -8708.395,E2 -8708.395} C_VEL
LIN {X 0,Y 447.702,Z 564.988,A -85,B 0,C 180,E1 -8711.228,E2 -8711.228} C_VEL
LIN {X 0,Y 447.476,Z 570.768,A -85,B 0,C 180,E1 -8712.188,E2 -8712.188} C_VEL
LIN {X 0,Y 450.724,Z 594.052,A -85,B 0,C 180,E1 -8712.705,E2 -8712.705} C_VEL
LIN {X 0,Y 449.844,Z 679.97,A -85,B 0,C 180,E1 -8714.133,E2 -8714.133} C_VEL
LIN {X 0,Y 449.385,Z 693.731,A -85,B 0,C 180,E1 -8714.553,E2 -8714.553} C_VEL
LIN {X 0,Y 448.872,Z 706.642,A -85,B 0,C 180,E1 -8715.145,E2 -8715.145} C_VEL
LIN {X 0,Y 448.196,Z 719.22,A -85,B 0,C 180,E1 -8715.934,E2 -8715.934} C_VEL
LIN {X 0,Y 447.621,Z 730.551,A -85,B 0,C 180,E1 -8716.849,E2 -8716.849} C_VEL
LIN {X 0,Y 447.083,Z 741.563,A -85,B 0,C 180,E1 -8717.978,E2 -8717.978} C_VEL
LIN {X 0,Y 446.516,Z 750.549,A -85,B 0,C 180,E1 -8719.113,E2 -8719.113} C_VEL
LIN {X 0,Y 446.063,Z 759.331,A -85,B 0,C 180,E1 -8720.478,E2 -8720.478} C_VEL
LIN {X 0,Y 445.766,Z 766.335,A -85,B 0,C 180,E1 -8721.843,E2 -8721.843} C_VEL
LIN {X 0,Y 445.555,Z 772.106,A -85,B 0,C 180,E1 -8723.252,E2 -8723.252} C_VEL
LIN {X 0,Y 445.488,Z 777.59,A -85,B 0,C 180,E1 -8725.022,E2 -8725.022} C_VEL
LIN {X 0,Y 445.425,Z 780.557,A -85,B 0,C 180,E1 -8726.382,E2 -8726.382} C_VEL
LIN {X 0,Y 445.467,Z 781.976,A -85,B 0,C 180,E1 -8727.287,E2 -8727.287} C_VEL
LIN {X 0,Y 445.45,Z 782.979,A -85,B 0,C 180,E1 -8728.192,E2 -8728.192} C_VEL
LIN {X 0,Y 445.427,Z 783.587,A -85,B 0,C 180,E1 -8729.096,E2 -8729.096} C_VEL
LIN {X 0,Y 445.4,Z 783.797,A -85,B 0,C 180,E1 -8730,E2 -8730} C_VEL
LIN {X 0,Y 445.427,Z 783.571,A -85,B 0,C 180,E1 -8730.904,E2 -8730.904} C_VEL
LIN {X 0,Y 445.45,Z 782.943,A -85,B 0,C 180,E1 -8731.808,E2 -8731.808} C_VEL
LIN {X 0,Y 445.467,Z 781.921,A -85,B 0,C 180,E1 -8732.713,E2 -8732.713} C_VEL
LIN {X 0,Y 445.425,Z 780.488,A -85,B 0,C 180,E1 -8733.618,E2 -8733.618} C_VEL
LIN {X 0,Y 445.488,Z 777.49,A -85,B 0,C 180,E1 -8734.978,E2 -8734.978} C_VEL
LIN {X 0,Y 445.558,Z 771.978,A -85,B 0,C 180,E1 -8736.748,E2 -8736.748} C_VEL
LIN {X 0,Y 445.764,Z 766.188,A -85,B 0,C 180,E1 -8738.157,E2 -8738.157} C_VEL
LIN {X 0,Y 446.059,Z 759.174,A -85,B 0,C 180,E1 -8739.522,E2 -8739.522} C_VEL
LIN {X 0,Y 446.511,Z 750.401,A -85,B 0,C 180,E1 -8740.887,E2 -8740.887} C_VEL
LIN {X 0,Y 447.044,Z 741.423,A -85,B 0,C 180,E1 -8742.023,E2 -8742.023} C_VEL
LIN {X 0,Y 447.607,Z 730.544,A -85,B 0,C 180,E1 -8743.143,E2 -8743.143} C_VEL
LIN {X 0,Y 448.214,Z 719.202,A -85,B 0,C 180,E1 -8744.066,E2 -8744.066} C_VEL
LIN {X 0,Y 448.865,Z 706.708,A -85,B 0,C 180,E1 -8744.855,E2 -8744.855} C_VEL
LIN {X 0,Y 449.403,Z 694.832,A -85,B 0,C 180,E1 -8745.417,E2 -8745.417} C_VEL
LIN {X 0,Y 449.782,Z 683.049,A -85,B 0,C 180,E1 -8745.811,E2 -8745.811} C_VEL
LIN {X 0,Y 450.11,Z 667.392,A -85,B 0,C 180,E1 -8746.119,E2 -8746.119} C_VEL
LIN {X 0,Y 450.727,Z 592.86,A -85,B 0,C 180,E1 -8747.346,E2 -8747.346} C_VEL
LIN {X 0,Y 447.443,Z 569.599,A -85,B 0,C 180,E1 -8747.898,E2 -8747.898} C_VEL
LIN {X 0,Y 448.316,Z 550.78,A -85,B 0,C 180,E1 -8751.134,E2 -8751.134} C_VEL
LIN {X 0,Y 449.379,Z 531.615,A -85,B 0,C 180,E1 -8754.482,E2 -8754.482} C_VEL
LIN {X 0,Y 449.279,Z 527.501,A -85,B 0,C 180,E1 -8755.23,E2 -8755.23} C_VEL
LIN {X 0,Y 446.751,Z 515.09,A -85,B 0,C 180,E1 -8757.65,E2 -8757.65} C_VEL
LIN {X 0,Y 446.499,Z 513.868,A -85,B 0,C 180,E1 -8757.921,E2 -8757.921} C_VEL
LIN {X 0,Y 446.417,Z 513.879,A -85,B 0,C 180,E1 -8761.299,E2 -8761.299} C_VEL
LIN {X 0,Y 446.43,Z 513.881,A -85,B 0,C 180,E1 -8764.522,E2 -8764.522} C_VEL
LIN {X 0,Y 446.436,Z 513.874,A -85,B 0,C 180,E1 -8768.082,E2 -8768.082} C_VEL
LIN {X 0,Y 446.446,Z 513.875,A -85,B 0,C 180,E1 -8770.92,E2 -8770.92} C_VEL
LIN {X 0,Y 446.443,Z 513.871,A -85,B 0,C 180,E1 -8773.84,E2 -8773.84} C_VEL
LIN {X 0,Y 446.418,Z 513.877,A -85,B 0,C 180,E1 -8776.399,E2 -8776.399} C_VEL
LIN {X 0,Y 446.444,Z 513.87,A -85,B 0,C 180,E1 -8779.802,E2 -8779.802} C_VEL
LIN {X 0,Y 446.424,Z 513.874,A -85,B 0,C 180,E1 -8782.122,E2 -8782.122} C_VEL
LIN {X 0,Y 446.425,Z 513.871,A -85,B 0,C 180,E1 -8785.476,E2 -8785.476} C_VEL
LIN {X 0,Y 446.414,Z 513.878,A -85,B 0,C 180,E1 -8788.699,E2 -8788.699} C_VEL
LIN {X 0,Y 446.478,Z 513.865,A -85,B 0,C 180,E1 -8791.82,E2 -8791.82} C_VEL
LIN {X 0,Y 446.452,Z 513.873,A -85,B 0,C 180,E1 -8794.847,E2 -8794.847} C_VEL
LIN {X 0,Y 446.44,Z 513.872,A -85,B 0,C 180,E1 -8798.244,E2 -8798.244} C_VEL
LIN {X 0,Y 446.449,Z 513.869,A -85,B 0,C 180,E1 -8801.648,E2 -8801.648} C_VEL
LIN {X 0,Y 446.499,Z 513.865,A -85,B 0,C 180,E1 -8804.479,E2 -8804.479} C_VEL
LIN {X 0,Y 446.507,Z 513.865,A -85,B 0,C 180,E1 -8807.383,E2 -8807.383} C_VEL
LIN {X 0,Y 446.53,Z 513.863,A -85,B 0,C 180,E1 -8810.944,E2 -8810.944} C_VEL
LIN {X 0,Y 446.643,Z 513.843,A -85,B 0,C 180,E1 -8813.676,E2 -8813.676} C_VEL
LIN {X 0,Y 446.701,Z 513.841,A -85,B 0,C 180,E1 -8817.294,E2 -8817.294} C_VEL
LIN {X 0,Y 446.785,Z 513.826,A -85,B 0,C 180,E1 -8820,E2 -8820} C_VEL
LIN {X 0,Y 446.702,Z 513.843,A -85,B 0,C 180,E1 -8822.705,E2 -8822.705} C_VEL
LIN {X 0,Y 446.643,Z 513.845,A -85,B 0,C 180,E1 -8826.323,E2 -8826.323} C_VEL
LIN {X 0,Y 446.529,Z 513.864,A -85,B 0,C 180,E1 -8829.055,E2 -8829.055} C_VEL
LIN {X 0,Y 446.514,Z 513.866,A -85,B 0,C 180,E1 -8832.729,E2 -8832.729} C_VEL
LIN {X 0,Y 446.486,Z 513.866,A -85,B 0,C 180,E1 -8836.228,E2 -8836.228} C_VEL
LIN {X 0,Y 446.46,Z 513.874,A -85,B 0,C 180,E1 -8839.303,E2 -8839.303} C_VEL
LIN {X 0,Y 446.408,Z 513.877,A -85,B 0,C 180,E1 -8842.2,E2 -8842.2} C_VEL
LIN {X 0,Y 446.448,Z 513.877,A -85,B 0,C 180,E1 -8845.152,E2 -8845.152} C_VEL
LIN {X 0,Y 446.475,Z 513.872,A -85,B 0,C 180,E1 -8848.179,E2 -8848.179} C_VEL
LIN {X 0,Y 446.525,Z 513.998,A -85,B 0,C 180,E1 -8851.756,E2 -8851.756} C_VEL
LIN {X 0,Y 447.867,Z 522.522,A -85,B 0,C 180,E1 -8853.947,E2 -8853.947} C_VEL
LIN {X 0,Y 447.877,Z 523.908,A -85,B 0,C 180,E1 -8854.227,E2 -8854.227} C_VEL
LIN {X 0,Y 451.191,Z 539.125,A -85,B 0,C 180,E1 -8854.631,E2 -8854.631} C_VEL
LIN {X 0,Y 450.152,Z 629.878,A -85,B 0,C 180,E1 -8856.147,E2 -8856.147} C_VEL
LIN {X 0,Y 449.803,Z 642.97,A -85,B 0,C 180,E1 -8856.544,E2 -8856.544} C_VEL
LIN {X 0,Y 449.484,Z 655.596,A -85,B 0,C 180,E1 -8857.117,E2 -8857.117} C_VEL
LIN {X 0,Y 448.964,Z 667.284,A -85,B 0,C 180,E1 -8857.834,E2 -8857.834} C_VEL
LIN {X 0,Y 448.436,Z 678.343,A -85,B 0,C 180,E1 -8858.707,E2 -8858.707} C_VEL
LIN {X 0,Y 447.851,Z 688.846,A -85,B 0,C 180,E1 -8859.743,E2 -8859.743} C_VEL
LIN {X 0,Y 447.262,Z 698.025,A -85,B 0,C 180,E1 -8860.861,E2 -8860.861} C_VEL
LIN {X 0,Y 446.766,Z 706.051,A -85,B 0,C 180,E1 -8862.063,E2 -8862.063} C_VEL
LIN {X 0,Y 446.329,Z 714.221,A -85,B 0,C 180,E1 -8863.589,E2 -8863.589} C_VEL
LIN {X 0,Y 446.008,Z 719.556,A -85,B 0,C 180,E1 -8864.84,E2 -8864.84} C_VEL
LIN {X 0,Y 445.793,Z 723.803,A -85,B 0,C 180,E1 -8866.08,E2 -8866.08} C_VEL
LIN {X 0,Y 445.667,Z 727.107,A -85,B 0,C 180,E1 -8867.306,E2 -8867.306} C_VEL
LIN {X 0,Y 445.495,Z 729.565,A -85,B 0,C 180,E1 -8868.504,E2 -8868.504} C_VEL
LIN {X 0,Y 445.366,Z 731.231,A -85,B 0,C 180,E1 -8869.686,E2 -8869.686} C_VEL
LIN {X 0,Y 445.319,Z 732.204,A -85,B 0,C 180,E1 -8870.857,E2 -8870.857} C_VEL
LIN {X 0,Y 445.322,Z 732.536,A -85,B 0,C 180,E1 -8872.1,E2 -8872.1} C_VEL
LIN {X 0,Y 445.326,Z 731.917,A -85,B 0,C 180,E1 -8873.596,E2 -8873.596} C_VEL
LIN {X 0,Y 445.411,Z 730.141,A -85,B 0,C 180,E1 -8875.133,E2 -8875.133} C_VEL
LIN {X 0,Y 445.624,Z 727.083,A -85,B 0,C 180,E1 -8876.706,E2 -8876.706} C_VEL
LIN {X 0,Y 445.825,Z 722.477,A -85,B 0,C 180,E1 -8878.348,E2 -8878.348} C_VEL
LIN {X 0,Y 446.122,Z 717.305,A -85,B 0,C 180,E1 -8879.728,E2 -8879.728} C_VEL
LIN {X 0,Y 446.471,Z 711.073,A -85,B 0,C 180,E1 -8881.051,E2 -8881.051} C_VEL
LIN {X 0,Y 446.905,Z 703.433,A -85,B 0,C 180,E1 -8882.361,E2 -8882.361} C_VEL
LIN {X 0,Y 447.372,Z 694.822,A -85,B 0,C 180,E1 -8883.564,E2 -8883.564} C_VEL
LIN {X 0,Y 447.955,Z 684.915,A -85,B 0,C 180,E1 -8884.69,E2 -8884.69} C_VEL
LIN {X 0,Y 448.536,Z 673.851,A -85,B 0,C 180,E1 -8885.691,E2 -8885.691} C_VEL
LIN {X 0,Y 448.744,Z 669.508,A -85,B 0,C 180,E1 -8886.027,E2 -8886.027} C_VEL
LIN {X 0,Y 448.218,Z 664.425,A -85,B 0,C 180,E1 -8886.408,E2 -8886.408} C_VEL
LIN {X 0,Y 445.669,Z 656.007,A -85,B 0,C 180,E1 -8887.018,E2 -8887.018} C_VEL
LIN {X 0,Y 443.251,Z 647.334,A -85,B 0,C 180,E1 -8887.539,E2 -8887.539} C_VEL
LIN {X 0,Y 442.925,Z 641.782,A -85,B 0,C 180,E1 -8887.779,E2 -8887.779} C_VEL
LIN {X 0,Y 443.184,Z 629.439,A -85,B 0,C 180,E1 -8888.151,E2 -8888.151} C_VEL
LIN {X 0,Y 444.101,Z 538.75,A -85,B 0,C 180,E1 -8889.684,E2 -8889.684} C_VEL
LIN {X 0,Y 440.662,Z 523.041,A -85,B 0,C 180,E1 -8890.106,E2 -8890.106} C_VEL
LIN {X 0,Y 439.724,Z 516.109,A -85,B 0,C 180,E1 -8891.841,E2 -8891.841} C_VEL
LIN {X 0,Y 439.444,Z 514.749,A -85,B 0,C 180,E1 -8892.19,E2 -8892.19} C_VEL
LIN {X 0,Y 439.445,Z 514.745,A -85,B 0,C 180,E1 -8895.174,E2 -8895.174} C_VEL
LIN {X 0,Y 439.48,Z 514.737,A -85,B 0,C 180,E1 -8898.002,E2 -8898.002} C_VEL
LIN {X 0,Y 439.545,Z 514.729,A -85,B 0,C 180,E1 -8901.726,E2 -8901.726} C_VEL
LIN {X 0,Y 439.615,Z 514.723,A -85,B 0,C 180,E1 -8904.496,E2 -8904.496} C_VEL
LIN {X 0,Y 439.633,Z 514.718,A -85,B 0,C 180,E1 -8908.168,E2 -8908.168} C_VEL
LIN {X 0,Y 439.761,Z 514.702,A -85,B 0,C 180,E1 -8910,E2 -8910} C_VEL
LIN {X 0,Y 439.653,Z 514.721,A -85,B 0,C 180,E1 -8912.749,E2 -8912.749} C_VEL
LIN {X 0,Y 439.616,Z 514.722,A -85,B 0,C 180,E1 -8916.425,E2 -8916.425} C_VEL
LIN {X 0,Y 439.497,Z 514.739,A -85,B 0,C 180,E1 -8919.201,E2 -8919.201} C_VEL
LIN {X 0,Y 439.463,Z 514.747,A -85,B 0,C 180,E1 -8922.937,E2 -8922.937} C_VEL
LIN {X 0,Y 439.444,Z 514.742,A -85,B 0,C 180,E1 -8926.349,E2 -8926.349} C_VEL
LIN {X 0,Y 439.399,Z 514.748,A -85,B 0,C 180,E1 -8929.626,E2 -8929.626} C_VEL
LIN {X 0,Y 439.361,Z 514.755,A -85,B 0,C 180,E1 -8932.575,E2 -8932.575} C_VEL
LIN {X 0,Y 439.4,Z 514.748,A -85,B 0,C 180,E1 -8935.584,E2 -8935.584} C_VEL
LIN {X 0,Y 439.42,Z 514.748,A -85,B 0,C 180,E1 -8938.672,E2 -8938.672} C_VEL
LIN {X 0,Y 439.379,Z 514.749,A -85,B 0,C 180,E1 -8942.033,E2 -8942.033} C_VEL
LIN {X 0,Y 439.39,Z 514.752,A -85,B 0,C 180,E1 -8945.34,E2 -8945.34} C_VEL
LIN {X 0,Y 439.393,Z 514.75,A -85,B 0,C 180,E1 -8948.593,E2 -8948.593} C_VEL
LIN {X 0,Y 439.398,Z 514.752,A -85,B 0,C 180,E1 -8951.259,E2 -8951.259} C_VEL
LIN {X 0,Y 439.403,Z 514.75,A -85,B 0,C 180,E1 -8954.728,E2 -8954.728} C_VEL
LIN {X 0,Y 439.404,Z 514.747,A -85,B 0,C 180,E1 -8957.797,E2 -8957.797} C_VEL
LIN {X 0,Y 439.444,Z 514.742,A -85,B 0,C 180,E1 -8960.23,E2 -8960.23} C_VEL
LIN {X 0,Y 439.369,Z 514.752,A -85,B 0,C 180,E1 -8963.713,E2 -8963.713} C_VEL
LIN {X 0,Y 439.364,Z 514.759,A -85,B 0,C 180,E1 -8967.054,E2 -8967.054} C_VEL
LIN {X 0,Y 439.387,Z 514.749,A -85,B 0,C 180,E1 -8970.275,E2 -8970.275} C_VEL
LIN {X 0,Y 439.424,Z 514.746,A -85,B 0,C 180,E1 -8973.589,E2 -8973.589} C_VEL
LIN {X 0,Y 439.377,Z 514.75,A -85,B 0,C 180,E1 -8976.43,E2 -8976.43} C_VEL
LIN {X 0,Y 439.379,Z 514.754,A -85,B 0,C 180,E1 -8979.397,E2 -8979.397} C_VEL
LIN {X 0,Y 439.421,Z 514.744,A -85,B 0,C 180,E1 -8982.31,E2 -8982.31} C_VEL
LIN {X 0,Y 439.437,Z 514.75,A -85,B 0,C 180,E1 -8985.174,E2 -8985.174} C_VEL
LIN {X 0,Y 439.499,Z 514.735,A -85,B 0,C 180,E1 -8988.002,E2 -8988.002} C_VEL
LIN {X 0,Y 439.539,Z 514.731,A -85,B 0,C 180,E1 -8991.727,E2 -8991.727} C_VEL
LIN {X 0,Y 439.619,Z 514.72,A -85,B 0,C 180,E1 -8994.496,E2 -8994.496} C_VEL
LIN {X 0,Y 439.627,Z 514.718,A -85,B 0,C 180,E1 -8998.168,E2 -8998.168} C_VEL
LIN {X 0,Y 439.755,Z 514.703,A -85,B 0,C 180,E1 -9000,E2 -9000} C_VEL
LIN {X 0,Y 439.656,Z 514.717,A -85,B 0,C 180,E1 -9002.749,E2 -9002.749} C_VEL
LIN {X 0,Y 439.614,Z 514.72,A -85,B 0,C 180,E1 -9006.426,E2 -9006.426} C_VEL
LIN {X 0,Y 439.492,Z 514.743,A -85,B 0,C 180,E1 -9009.202,E2 -9009.202} C_VEL
LIN {X 0,Y 439.461,Z 514.743,A -85,B 0,C 180,E1 -9012.938,E2 -9012.938} C_VEL
LIN {X 0,Y 439.439,Z 514.742,A -85,B 0,C 180,E1 -9016.349,E2 -9016.349} C_VEL
LIN {X 0,Y 439.395,Z 514.751,A -85,B 0,C 180,E1 -9019.627,E2 -9019.627} C_VEL
LIN {X 0,Y 439.358,Z 514.753,A -85,B 0,C 180,E1 -9022.576,E2 -9022.576} C_VEL
LIN {X 0,Y 439.399,Z 514.751,A -85,B 0,C 180,E1 -9025.586,E2 -9025.586} C_VEL
LIN {X 0,Y 439.419,Z 514.745,A -85,B 0,C 180,E1 -9028.674,E2 -9028.674} C_VEL
LIN {X 0,Y 439.379,Z 514.75,A -85,B 0,C 180,E1 -9032.034,E2 -9032.034} C_VEL
LIN {X 0,Y 439.391,Z 514.756,A -85,B 0,C 180,E1 -9035.342,E2 -9035.342} C_VEL
LIN {X 0,Y 439.386,Z 514.749,A -85,B 0,C 180,E1 -9038.595,E2 -9038.595} C_VEL
LIN {X 0,Y 439.386,Z 514.756,A -85,B 0,C 180,E1 -9041.258,E2 -9041.258} C_VEL
LIN {X 0,Y 439.404,Z 514.747,A -85,B 0,C 180,E1 -9044.729,E2 -9044.729} C_VEL
LIN {X 0,Y 439.41,Z 514.748,A -85,B 0,C 180,E1 -9047.799,E2 -9047.799} C_VEL
LIN {X 0,Y 439.449,Z 514.741,A -85,B 0,C 180,E1 -9050.231,E2 -9050.231} C_VEL
LIN {X 0,Y 439.376,Z 514.753,A -85,B 0,C 180,E1 -9053.714,E2 -9053.714} C_VEL
LIN {X 0,Y 439.373,Z 514.757,A -85,B 0,C 180,E1 -9057.055,E2 -9057.055} C_VEL
LIN {X 0,Y 439.383,Z 514.754,A -85,B 0,C 180,E1 -9060.275,E2 -9060.275} C_VEL
LIN {X 0,Y 439.471,Z 514.833,A -85,B 0,C 180,E1 -9061.846,E2 -9061.846} C_VEL
LIN {X 0,Y 442.338,Z 528.848,A -85,B 0,C 180,E1 -9064.598,E2 -9064.598} C_VEL
LIN {X 0,Y 442.557,Z 533.235,A -85,B 0,C 180,E1 -9065.406,E2 -9065.406} C_VEL
LIN {X 0,Y 441.406,Z 552.224,A -85,B 0,C 180,E1 -9068.764,E2 -9068.764} C_VEL
LIN {X 0,Y 440.479,Z 570.171,A -85,B 0,C 180,E1 -9071.895,E2 -9071.895} C_VEL
LIN {X 0,Y 443.929,Z 595.178,A -85,B 0,C 180,E1 -9072.468,E2 -9072.468} C_VEL
LIN {X 0,Y 443.018,Z 679.106,A -85,B 0,C 180,E1 -9073.882,E2 -9073.882} C_VEL
LIN {X 0,Y 442.599,Z 692.259,A -85,B 0,C 180,E1 -9074.281,E2 -9074.281} C_VEL
LIN {X 0,Y 442.068,Z 703.824,A -85,B 0,C 180,E1 -9074.793,E2 -9074.793} C_VEL
LIN {X 0,Y 441.476,Z 715.422,A -85,B 0,C 180,E1 -9075.48,E2 -9075.48} C_VEL
LIN {X 0,Y 440.862,Z 727.258,A -85,B 0,C 180,E1 -9076.394,E2 -9076.394} C_VEL
LIN {X 0,Y 440.189,Z 737.972,A -85,B 0,C 180,E1 -9077.436,E2 -9077.436} C_VEL
LIN {X 0,Y 439.707,Z 746.683,A -85,B 0,C 180,E1 -9078.475,E2 -9078.475} C_VEL
LIN {X 0,Y 439.216,Z 754.707,A -85,B 0,C 180,E1 -9079.63,E2 -9079.63} C_VEL
LIN {X 0,Y 438.832,Z 762.566,A -85,B 0,C 180,E1 -9081.017,E2 -9081.017} C_VEL
LIN {X 0,Y 438.539,Z 769.771,A -85,B 0,C 180,E1 -9082.634,E2 -9082.634} C_VEL
LIN {X 0,Y 438.393,Z 774.418,A -85,B 0,C 180,E1 -9083.969,E2 -9083.969} C_VEL
LIN {X 0,Y 438.354,Z 778.245,A -85,B 0,C 180,E1 -9085.402,E2 -9085.402} C_VEL
LIN {X 0,Y 438.328,Z 780.138,A -85,B 0,C 180,E1 -9086.323,E2 -9086.323} C_VEL
LIN {X 0,Y 438.392,Z 781.563,A -85,B 0,C 180,E1 -9087.243,E2 -9087.243} C_VEL
LIN {X 0,Y 438.366,Z 782.567,A -85,B 0,C 180,E1 -9088.163,E2 -9088.163} C_VEL
LIN {X 0,Y 438.366,Z 783.178,A -85,B 0,C 180,E1 -9089.081,E2 -9089.081} C_VEL
LIN {X 0,Y 438.338,Z 783.39,A -85,B 0,C 180,E1 -9090,E2 -9090} C_VEL
LIN {X 0,Y 438.366,Z 783.166,A -85,B 0,C 180,E1 -9090.919,E2 -9090.919} C_VEL
LIN {X 0,Y 438.392,Z 781.516,A -85,B 0,C 180,E1 -9092.757,E2 -9092.757} C_VEL
LIN {X 0,Y 438.328,Z 780.082,A -85,B 0,C 180,E1 -9093.677,E2 -9093.677} C_VEL
LIN {X 0,Y 438.419,Z 777.086,A -85,B 0,C 180,E1 -9095.058,E2 -9095.058} C_VEL
LIN {X 0,Y 438.449,Z 773.031,A -85,B 0,C 180,E1 -9096.442,E2 -9096.442} C_VEL
LIN {X 0,Y 438.667,Z 766.81,A -85,B 0,C 180,E1 -9098.058,E2 -9098.058} C_VEL
LIN {X 0,Y 438.963,Z 760.022,A -85,B 0,C 180,E1 -9099.445,E2 -9099.445} C_VEL
LIN {X 0,Y 439.384,Z 751.61,A -85,B 0,C 180,E1 -9100.832,E2 -9100.832} C_VEL
LIN {X 0,Y 439.947,Z 742.99,A -85,B 0,C 180,E1 -9101.986,E2 -9101.986} C_VEL
LIN {X 0,Y 440.559,Z 732.176,A -85,B 0,C 180,E1 -9103.156,E2 -9103.156} C_VEL
LIN {X 0,Y 441.239,Z 720.382,A -85,B 0,C 180,E1 -9104.175,E2 -9104.175} C_VEL
LIN {X 0,Y 441.867,Z 708.308,A -85,B 0,C 180,E1 -9104.978,E2 -9104.978} C_VEL
LIN {X 0,Y 442.493,Z 695.767,A -85,B 0,C 180,E1 -9105.605,E2 -9105.605} C_VEL
LIN {X 0,Y 442.905,Z 683.753,A -85,B 0,C 180,E1 -9106.033,E2 -9106.033} C_VEL
LIN {X 0,Y 443.295,Z 668.951,A -85,B 0,C 180,E1 -9106.344,E2 -9106.344} C_VEL
LIN {X 0,Y 443.949,Z 593.482,A -85,B 0,C 180,E1 -9107.611,E2 -9107.611} C_VEL
LIN {X 0,Y 440.479,Z 569.276,A -85,B 0,C 180,E1 -9108.184,E2 -9108.184} C_VEL
LIN {X 0,Y 441.527,Z 549.057,A -85,B 0,C 180,E1 -9111.72,E2 -9111.72} C_VEL
LIN {X 0,Y 442.547,Z 531.829,A -85,B 0,C 180,E1 -9114.792,E2 -9114.792} C_VEL
LIN {X 0,Y 442.042,Z 527.197,A -85,B 0,C 180,E1 -9115.673,E2 -9115.673} C_VEL
LIN {X 0,Y 439.462,Z 514.746,A -85,B 0,C 180,E1 -9118.181,E2 -9118.181} C_VEL
LIN {X 0,Y 439.374,Z 514.756,A -85,B 0,C 180,E1 -9121.86,E2 -9121.86} C_VEL
LIN {X 0,Y 439.4,Z 514.754,A -85,B 0,C 180,E1 -9125.155,E2 -9125.155} C_VEL
LIN {X 0,Y 439.396,Z 514.755,A -85,B 0,C 180,E1 -9128.592,E2 -9128.592} C_VEL
LIN {X 0,Y 439.403,Z 514.75,A -85,B 0,C 180,E1 -9131.258,E2 -9131.258} C_VEL
LIN {X 0,Y 439.407,Z 514.752,A -85,B 0,C 180,E1 -9134.727,E2 -9134.727} C_VEL
LIN {X 0,Y 439.394,Z 514.746,A -85,B 0,C 180,E1 -9137.795,E2 -9137.795} C_VEL
LIN {X 0,Y 439.426,Z 514.746,A -85,B 0,C 180,E1 -9140.227,E2 -9140.227} C_VEL
LIN {X 0,Y 439.373,Z 514.751,A -85,B 0,C 180,E1 -9143.712,E2 -9143.712} C_VEL
LIN {X 0,Y 439.368,Z 514.757,A -85,B 0,C 180,E1 -9147.053,E2 -9147.053} C_VEL
LIN {X 0,Y 439.391,Z 514.75,A -85,B 0,C 180,E1 -9150.274,E2 -9150.274} C_VEL
LIN {X 0,Y 439.427,Z 514.745,A -85,B 0,C 180,E1 -9153.588,E2 -9153.588} C_VEL
LIN {X 0,Y 439.379,Z 514.749,A -85,B 0,C 180,E1 -9156.429,E2 -9156.429} C_VEL
LIN {X 0,Y 439.381,Z 514.75,A -85,B 0,C 180,E1 -9159.396,E2 -9159.396} C_VEL
LIN {X 0,Y 439.424,Z 514.745,A -85,B 0,C 180,E1 -9162.309,E2 -9162.309} C_VEL
LIN {X 0,Y 439.441,Z 514.746,A -85,B 0,C 180,E1 -9165.173,E2 -9165.173} C_VEL
LIN {X 0,Y 439.476,Z 514.738,A -85,B 0,C 180,E1 -9168.001,E2 -9168.001} C_VEL
LIN {X 0,Y 439.539,Z 514.731,A -85,B 0,C 180,E1 -9171.726,E2 -9171.726} C_VEL
LIN {X 0,Y 439.619,Z 514.719,A -85,B 0,C 180,E1 -9174.495,E2 -9174.495} C_VEL
LIN {X 0,Y 439.627,Z 514.719,A -85,B 0,C 180,E1 -9178.167,E2 -9178.167} C_VEL
LIN {X 0,Y 439.755,Z 514.702,A -85,B 0,C 180,E1 -9180,E2 -9180} C_VEL
LIN {X 0,Y 439.649,Z 514.722,A -85,B 0,C 180,E1 -9182.748,E2 -9182.748} C_VEL
LIN {X 0,Y 439.613,Z 514.721,A -85,B 0,C 180,E1 -9186.425,E2 -9186.425} C_VEL
LIN {X 0,Y 439.491,Z 514.741,A -85,B 0,C 180,E1 -9189.201,E2 -9189.201} C_VEL
LIN {X 0,Y 439.459,Z 514.747,A -85,B 0,C 180,E1 -9192.937,E2 -9192.937} C_VEL
LIN {X 0,Y 439.437,Z 514.745,A -85,B 0,C 180,E1 -9196.349,E2 -9196.349} C_VEL
LIN {X 0,Y 439.393,Z 514.752,A -85,B 0,C 180,E1 -9199.626,E2 -9199.626} C_VEL
LIN {X 0,Y 439.355,Z 514.757,A -85,B 0,C 180,E1 -9202.575,E2 -9202.575} C_VEL
LIN {X 0,Y 439.396,Z 514.758,A -85,B 0,C 180,E1 -9205.585,E2 -9205.585} C_VEL
LIN {X 0,Y 439.416,Z 514.752,A -85,B 0,C 180,E1 -9208.673,E2 -9208.673} C_VEL
LIN {X 0,Y 439.474,Z 514.844,A -85,B 0,C 180,E1 -9211.515,E2 -9211.515} C_VEL
LIN {X 0,Y 440.908,Z 522.933,A -85,B 0,C 180,E1 -9213.635,E2 -9213.635} C_VEL
LIN {X 0,Y 440.938,Z 524.02,A -85,B 0,C 180,E1 -9213.907,E2 -9213.907} C_VEL
LIN {X 0,Y 444.457,Z 540.146,A -85,B 0,C 180,E1 -9214.358,E2 -9214.358} C_VEL
LIN {X 0,Y 443.358,Z 630.34,A -85,B 0,C 180,E1 -9215.892,E2 -9215.892} C_VEL
LIN {X 0,Y 443.007,Z 644.178,A -85,B 0,C 180,E1 -9216.326,E2 -9216.326} C_VEL
LIN {X 0,Y 442.643,Z 656.438,A -85,B 0,C 180,E1 -9216.899,E2 -9216.899} C_VEL
LIN {X 0,Y 442.142,Z 667.194,A -85,B 0,C 180,E1 -9217.567,E2 -9217.567} C_VEL
LIN {X 0,Y 441.591,Z 678.293,A -85,B 0,C 180,E1 -9218.45,E2 -9218.45} C_VEL
LIN {X 0,Y 440.905,Z 688.854,A -85,B 0,C 180,E1 -9219.497,E2 -9219.497} C_VEL
LIN {X 0,Y 440.318,Z 698.262,A -85,B 0,C 180,E1 -9220.653,E2 -9220.653} C_VEL
LIN {X 0,Y 439.74,Z 707.185,A -85,B 0,C 180,E1 -9222.023,E2 -9222.023} C_VEL
LIN {X 0,Y 439.302,Z 714.717,A -85,B 0,C 180,E1 -9223.465,E2 -9223.465} C_VEL
LIN {X 0,Y 438.977,Z 720.217,A -85,B 0,C 180,E1 -9224.783,E2 -9224.783} C_VEL
LIN {X 0,Y 438.674,Z 725.594,A -85,B 0,C 180,E1 -9226.458,E2 -9226.458} C_VEL
LIN {X 0,Y 438.56,Z 728.581,A -85,B 0,C 180,E1 -9227.698,E2 -9227.698} C_VEL
LIN {X 0,Y 438.358,Z 730.696,A -85,B 0,C 180,E1 -9228.904,E2 -9228.904} C_VEL
LIN {X 0,Y 438.237,Z 732.29,A -85,B 0,C 180,E1 -9230.333,E2 -9230.333} C_VEL
LIN {X 0,Y 438.223,Z 732.922,A -85,B 0,C 180,E1 -9231.797,E2 -9231.797} C_VEL
LIN {X 0,Y 438.239,Z 732.332,A -85,B 0,C 180,E1 -9233.605,E2 -9233.605} C_VEL
LIN {X 0,Y 438.301,Z 731.004,A -85,B 0,C 180,E1 -9234.861,E2 -9234.861} C_VEL
LIN {X 0,Y 438.522,Z 728.236,A -85,B 0,C 180,E1 -9236.447,E2 -9236.447} C_VEL
LIN {X 0,Y 438.719,Z 723.912,A -85,B 0,C 180,E1 -9238.105,E2 -9238.105} C_VEL
LIN {X 0,Y 439.025,Z 718.914,A -85,B 0,C 180,E1 -9239.535,E2 -9239.535} C_VEL
LIN {X 0,Y 439.416,Z 712.086,A -85,B 0,C 180,E1 -9241.066,E2 -9241.066} C_VEL
LIN {X 0,Y 439.87,Z 704.583,A -85,B 0,C 180,E1 -9242.398,E2 -9242.398} C_VEL
LIN {X 0,Y 440.412,Z 695.371,A -85,B 0,C 180,E1 -9243.716,E2 -9243.716} C_VEL
LIN {X 0,Y 441.04,Z 684.976,A -85,B 0,C 180,E1 -9244.914,E2 -9244.914} C_VEL
LIN {X 0,Y 441.67,Z 673.734,A -85,B 0,C 180,E1 -9245.937,E2 -9245.937} C_VEL
LIN {X 0,Y 442.183,Z 662.57,A -85,B 0,C 180,E1 -9246.744,E2 -9246.744} C_VEL
LIN {X 0,Y 442.643,Z 651.217,A -85,B 0,C 180,E1 -9247.379,E2 -9247.379} C_VEL
LIN {X 0,Y 442.925,Z 641.782,A -85,B 0,C 180,E1 -9247.779,E2 -9247.779} C_VEL
LIN {X 0,Y 442.89,Z 637.998,A -85,B 0,C 180,E1 -9247.918,E2 -9247.918} C_VEL
LIN {X 0,Y 441.81,Z 632.398,A -85,B 0,C 180,E1 -9248.127,E2 -9248.127} C_VEL
LIN {X 0,Y 437.219,Z 617.59,A -85,B 0,C 180,E1 -9248.6,E2 -9248.6} C_VEL
LIN {X 0,Y 436.614,Z 611.771,A -85,B 0,C 180,E1 -9248.721,E2 -9248.721} C_VEL
LIN {X 0,Y 437.423,Z 540.264,A -85,B 0,C 180,E1 -9249.932,E2 -9249.932} C_VEL
LIN {X 0,Y 433.642,Z 523.368,A -85,B 0,C 180,E1 -9250.411,E2 -9250.411} C_VEL
LIN {X 0,Y 432.417,Z 515.623,A -85,B 0,C 180,E1 -9252.411,E2 -9252.411} C_VEL
LIN {X 0,Y 432.393,Z 515.627,A -85,B 0,C 180,E1 -9254.927,E2 -9254.927} C_VEL
LIN {X 0,Y 432.456,Z 515.612,A -85,B 0,C 180,E1 -9257.804,E2 -9257.804} C_VEL
LIN {X 0,Y 432.489,Z 515.608,A -85,B 0,C 180,E1 -9261.59,E2 -9261.59} C_VEL
LIN {X 0,Y 432.591,Z 515.597,A -85,B 0,C 180,E1 -9264.406,E2 -9264.406} C_VEL
LIN {X 0,Y 432.603,Z 515.594,A -85,B 0,C 180,E1 -9268.138,E2 -9268.138} C_VEL
LIN {X 0,Y 432.731,Z 515.578,A -85,B 0,C 180,E1 -9270,E2 -9270} C_VEL
LIN {X 0,Y 432.602,Z 515.6,A -85,B 0,C 180,E1 -9272.793,E2 -9272.793} C_VEL
LIN {X 0,Y 432.571,Z 515.6,A -85,B 0,C 180,E1 -9276.53,E2 -9276.53} C_VEL
LIN {X 0,Y 432.44,Z 515.617,A -85,B 0,C 180,E1 -9279.353,E2 -9279.353} C_VEL
LIN {X 0,Y 432.428,Z 515.621,A -85,B 0,C 180,E1 -9282.803,E2 -9282.803} C_VEL
LIN {X 0,Y 432.409,Z 515.62,A -85,B 0,C 180,E1 -9286.479,E2 -9286.479} C_VEL
LIN {X 0,Y 432.335,Z 515.627,A -85,B 0,C 180,E1 -9289.96,E2 -9289.96} C_VEL
LIN {X 0,Y 432.315,Z 515.637,A -85,B 0,C 180,E1 -9292.964,E2 -9292.964} C_VEL
LIN {X 0,Y 432.359,Z 515.624,A -85,B 0,C 180,E1 -9296.032,E2 -9296.032} C_VEL
LIN {X 0,Y 432.348,Z 515.631,A -85,B 0,C 180,E1 -9299.186,E2 -9299.186} C_VEL
LIN {X 0,Y 432.327,Z 515.628,A -85,B 0,C 180,E1 -9302.294,E2 -9302.294} C_VEL
LIN {X 0,Y 432.335,Z 515.63,A -85,B 0,C 180,E1 -9304.677,E2 -9304.677} C_VEL
LIN {X 0,Y 432.347,Z 515.625,A -85,B 0,C 180,E1 -9308.148,E2 -9308.148} C_VEL
LIN {X 0,Y 432.366,Z 515.625,A -85,B 0,C 180,E1 -9311.608,E2 -9311.608} C_VEL
LIN {X 0,Y 432.371,Z 515.623,A -85,B 0,C 180,E1 -9314.341,E2 -9314.341} C_VEL
LIN {X 0,Y 432.358,Z 515.631,A -85,B 0,C 180,E1 -9317.009,E2 -9317.009} C_VEL
LIN {X 0,Y 432.35,Z 515.625,A -85,B 0,C 180,E1 -9319.817,E2 -9319.817} C_VEL
LIN {X 0,Y 432.309,Z 515.637,A -85,B 0,C 180,E1 -9323.023,E2 -9323.023} C_VEL
LIN {X 0,Y 432.351,Z 515.625,A -85,B 0,C 180,E1 -9325.996,E2 -9325.996} C_VEL
LIN {X 0,Y 432.386,Z 515.622,A -85,B 0,C 180,E1 -9329.744,E2 -9329.744} C_VEL
LIN {X 0,Y 432.391,Z 515.625,A -85,B 0,C 180,E1 -9333.372,E2 -9333.372} C_VEL
LIN {X 0,Y 432.362,Z 515.624,A -85,B 0,C 180,E1 -9336.023,E2 -9336.023} C_VEL
LIN {X 0,Y 432.341,Z 515.633,A -85,B 0,C 180,E1 -9339.046,E2 -9339.046} C_VEL
LIN {X 0,Y 432.368,Z 515.623,A -85,B 0,C 180,E1 -9342.011,E2 -9342.011} C_VEL
LIN {X 0,Y 432.385,Z 515.625,A -85,B 0,C 180,E1 -9344.927,E2 -9344.927} C_VEL
LIN {X 0,Y 432.472,Z 515.611,A -85,B 0,C 180,E1 -9347.804,E2 -9347.804} C_VEL
LIN {X 0,Y 432.483,Z 515.611,A -85,B 0,C 180,E1 -9351.591,E2 -9351.591} C_VEL
LIN {X 0,Y 432.595,Z 515.595,A -85,B 0,C 180,E1 -9354.407,E2 -9354.407} C_VEL
LIN {X 0,Y 432.597,Z 515.594,A -85,B 0,C 180,E1 -9358.138,E2 -9358.138} C_VEL
LIN {X 0,Y 432.725,Z 515.579,A -85,B 0,C 180,E1 -9360,E2 -9360} C_VEL
LIN {X 0,Y 432.605,Z 515.596,A -85,B 0,C 180,E1 -9362.794,E2 -9362.794} C_VEL
LIN {X 0,Y 432.568,Z 515.599,A -85,B 0,C 180,E1 -9366.531,E2 -9366.531} C_VEL
LIN {X 0,Y 432.436,Z 515.621,A -85,B 0,C 180,E1 -9369.354,E2 -9369.354} C_VEL
LIN {X 0,Y 432.424,Z 515.618,A -85,B 0,C 180,E1 -9372.805,E2 -9372.805} C_VEL
LIN {X 0,Y 432.405,Z 515.619,A -85,B 0,C 180,E1 -9376.48,E2 -9376.48} C_VEL
LIN {X 0,Y 432.331,Z 515.628,A -85,B 0,C 180,E1 -9379.961,E2 -9379.961} C_VEL
LIN {X 0,Y 432.312,Z 515.634,A -85,B 0,C 180,E1 -9382.965,E2 -9382.965} C_VEL
LIN {X 0,Y 432.358,Z 515.625,A -85,B 0,C 180,E1 -9386.033,E2 -9386.033} C_VEL
LIN {X 0,Y 432.347,Z 515.632,A -85,B 0,C 180,E1 -9389.188,E2 -9389.188} C_VEL
LIN {X 0,Y 432.327,Z 515.628,A -85,B 0,C 180,E1 -9392.296,E2 -9392.296} C_VEL
LIN {X 0,Y 432.336,Z 515.628,A -85,B 0,C 180,E1 -9394.678,E2 -9394.678} C_VEL
LIN {X 0,Y 432.343,Z 515.626,A -85,B 0,C 180,E1 -9398.15,E2 -9398.15} C_VEL
LIN {X 0,Y 432.331,Z 515.632,A -85,B 0,C 180,E1 -9401.603,E2 -9401.603} C_VEL
LIN {X 0,Y 432.338,Z 515.626,A -85,B 0,C 180,E1 -9404.347,E2 -9404.347} C_VEL
LIN {X 0,Y 432.364,Z 515.627,A -85,B 0,C 180,E1 -9407.01,E2 -9407.01} C_VEL
LIN {X 0,Y 432.356,Z 515.627,A -85,B 0,C 180,E1 -9409.818,E2 -9409.818} C_VEL
LIN {X 0,Y 432.315,Z 515.633,A -85,B 0,C 180,E1 -9413.024,E2 -9413.024} C_VEL
LIN {X 0,Y 432.359,Z 515.628,A -85,B 0,C 180,E1 -9415.997,E2 -9415.997} C_VEL
LIN {X 0,Y 432.348,Z 515.633,A -85,B 0,C 180,E1 -9419.49,E2 -9419.49} C_VEL
LIN {X 0,Y 432.418,Z 515.825,A -85,B 0,C 180,E1 -9421.621,E2 -9421.621} C_VEL
LIN {X 0,Y 435.056,Z 528.404,A -85,B 0,C 180,E1 -9424.141,E2 -9424.141} C_VEL
LIN {X 0,Y 435.666,Z 532.863,A -85,B 0,C 180,E1 -9425,E2 -9425} C_VEL
LIN {X 0,Y 434.516,Z 551.79,A -85,B 0,C 180,E1 -9428.41,E2 -9428.41} C_VEL
LIN {X 0,Y 433.529,Z 569.782,A -85,B 0,C 180,E1 -9431.604,E2 -9431.604} C_VEL
LIN {X 0,Y 437.118,Z 595.821,A -85,B 0,C 180,E1 -9432.213,E2 -9432.213} C_VEL
LIN {X 0,Y 436.155,Z 679.373,A -85,B 0,C 180,E1 -9433.652,E2 -9433.652} C_VEL
LIN {X 0,Y 435.665,Z 693.058,A -85,B 0,C 180,E1 -9434.084,E2 -9434.084} C_VEL
LIN {X 0,Y 435.106,Z 705.419,A -85,B 0,C 180,E1 -9434.663,E2 -9434.663} C_VEL
LIN {X 0,Y 434.385,Z 718.089,A -85,B 0,C 180,E1 -9435.477,E2 -9435.477} C_VEL
LIN {X 0,Y 433.807,Z 728.508,A -85,B 0,C 180,E1 -9436.333,E2 -9436.333} C_VEL
LIN {X 0,Y 433.151,Z 738.539,A -85,B 0,C 180,E1 -9437.348,E2 -9437.348} C_VEL
LIN {X 0,Y 432.594,Z 747.938,A -85,B 0,C 180,E1 -9438.521,E2 -9438.521} C_VEL
LIN {X 0,Y 432.022,Z 757.034,A -85,B 0,C 180,E1 -9439.929,E2 -9439.929} C_VEL
LIN {X 0,Y 431.694,Z 764.371,A -85,B 0,C 180,E1 -9441.339,E2 -9441.339} C_VEL
LIN {X 0,Y 431.466,Z 769.326,A -85,B 0,C 180,E1 -9442.513,E2 -9442.513} C_VEL
LIN {X 0,Y 431.294,Z 774.412,A -85,B 0,C 180,E1 -9444.009,E2 -9444.009} C_VEL
LIN {X 0,Y 431.286,Z 777.82,A -85,B 0,C 180,E1 -9445.327,E2 -9445.327} C_VEL
LIN {X 0,Y 431.232,Z 779.715,A -85,B 0,C 180,E1 -9446.262,E2 -9446.262} C_VEL
LIN {X 0,Y 431.318,Z 781.147,A -85,B 0,C 180,E1 -9447.198,E2 -9447.198} C_VEL
LIN {X 0,Y 431.285,Z 782.154,A -85,B 0,C 180,E1 -9448.132,E2 -9448.132} C_VEL
LIN {X 0,Y 431.277,Z 782.766,A -85,B 0,C 180,E1 -9449.066,E2 -9449.066} C_VEL
LIN {X 0,Y 431.278,Z 782.983,A -85,B 0,C 180,E1 -9450,E2 -9450} C_VEL
LIN {X 0,Y 431.277,Z 782.76,A -85,B 0,C 180,E1 -9450.934,E2 -9450.934} C_VEL
LIN {X 0,Y 431.285,Z 782.133,A -85,B 0,C 180,E1 -9451.868,E2 -9451.868} C_VEL
LIN {X 0,Y 431.318,Z 781.111,A -85,B 0,C 180,E1 -9452.802,E2 -9452.802} C_VEL
LIN {X 0,Y 431.232,Z 779.677,A -85,B 0,C 180,E1 -9453.738,E2 -9453.738} C_VEL
LIN {X 0,Y 431.325,Z 776.68,A -85,B 0,C 180,E1 -9455.141,E2 -9455.141} C_VEL
LIN {X 0,Y 431.377,Z 772.625,A -85,B 0,C 180,E1 -9456.548,E2 -9456.548} C_VEL
LIN {X 0,Y 431.596,Z 766.404,A -85,B 0,C 180,E1 -9458.191,E2 -9458.191} C_VEL
LIN {X 0,Y 431.905,Z 759.613,A -85,B 0,C 180,E1 -9459.601,E2 -9459.601} C_VEL
LIN {X 0,Y 432.384,Z 751.203,A -85,B 0,C 180,E1 -9461.01,E2 -9461.01} C_VEL
LIN {X 0,Y 432.943,Z 742.585,A -85,B 0,C 180,E1 -9462.182,E2 -9462.182} C_VEL
LIN {X 0,Y 433.544,Z 732.809,A -85,B 0,C 180,E1 -9463.27,E2 -9463.27} C_VEL
LIN {X 0,Y 434.249,Z 721.466,A -85,B 0,C 180,E1 -9464.288,E2 -9464.288} C_VEL
LIN {X 0,Y 434.898,Z 709.958,A -85,B 0,C 180,E1 -9465.104,E2 -9465.104} C_VEL
LIN {X 0,Y 435.474,Z 698.095,A -85,B 0,C 180,E1 -9465.743,E2 -9465.743} C_VEL
LIN {X 0,Y 436.053,Z 684.478,A -85,B 0,C 180,E1 -9466.262,E2 -9466.262} C_VEL
LIN {X 0,Y 436.397,Z 672.419,A -85,B 0,C 180,E1 -9466.549,E2 -9466.549} C_VEL
LIN {X 0,Y 437.239,Z 594.502,A -85,B 0,C 180,E1 -9467.877,E2 -9467.877} C_VEL
LIN {X 0,Y 433.522,Z 568.752,A -85,B 0,C 180,E1 -9468.514,E2 -9468.514} C_VEL
LIN {X 0,Y 434.634,Z 548.741,A -85,B 0,C 180,E1 -9472.083,E2 -9472.083} C_VEL
LIN {X 0,Y 435.623,Z 532.687,A -85,B 0,C 180,E1 -9474.998,E2 -9474.998} C_VEL
LIN {X 0,Y 434.784,Z 526.892,A -85,B 0,C 180,E1 -9476.134,E2 -9476.134} C_VEL
LIN {X 0,Y 432.389,Z 515.628,A -85,B 0,C 180,E1 -9478.468,E2 -9478.468} C_VEL
LIN {X 0,Y 432.322,Z 515.635,A -85,B 0,C 180,E1 -9481.345,E2 -9481.345} C_VEL
LIN {X 0,Y 432.341,Z 515.636,A -85,B 0,C 180,E1 -9484.676,E2 -9484.676} C_VEL
LIN {X 0,Y 432.351,Z 515.63,A -85,B 0,C 180,E1 -9488.147,E2 -9488.147} C_VEL
LIN {X 0,Y 432.371,Z 515.625,A -85,B 0,C 180,E1 -9491.607,E2 -9491.607} C_VEL
LIN {X 0,Y 432.376,Z 515.627,A -85,B 0,C 180,E1 -9494.34,E2 -9494.34} C_VEL
LIN {X 0,Y 432.331,Z 515.628,A -85,B 0,C 180,E1 -9498.202,E2 -9498.202} C_VEL
LIN {X 0,Y 432.347,Z 515.629,A -85,B 0,C 180,E1 -9501.283,E2 -9501.283} C_VEL
LIN {X 0,Y 432.341,Z 515.629,A -85,B 0,C 180,E1 -9504.367,E2 -9504.367} C_VEL
LIN {X 0,Y 432.318,Z 515.631,A -85,B 0,C 180,E1 -9507.556,E2 -9507.556} C_VEL
LIN {X 0,Y 432.389,Z 515.62,A -85,B 0,C 180,E1 -9509.743,E2 -9509.743} C_VEL
LIN {X 0,Y 432.394,Z 515.623,A -85,B 0,C 180,E1 -9513.371,E2 -9513.371} C_VEL
LIN {X 0,Y 432.364,Z 515.62,A -85,B 0,C 180,E1 -9516.023,E2 -9516.023} C_VEL
LIN {X 0,Y 432.343,Z 515.628,A -85,B 0,C 180,E1 -9519.045,E2 -9519.045} C_VEL
LIN {X 0,Y 432.37,Z 515.623,A -85,B 0,C 180,E1 -9522.01,E2 -9522.01} C_VEL
LIN {X 0,Y 432.389,Z 515.628,A -85,B 0,C 180,E1 -9524.926,E2 -9524.926} C_VEL
LIN {X 0,Y 432.451,Z 515.614,A -85,B 0,C 180,E1 -9527.803,E2 -9527.803} C_VEL
LIN {X 0,Y 432.483,Z 515.611,A -85,B 0,C 180,E1 -9531.59,E2 -9531.59} C_VEL
LIN {X 0,Y 432.595,Z 515.594,A -85,B 0,C 180,E1 -9534.406,E2 -9534.406} C_VEL
LIN {X 0,Y 432.597,Z 515.595,A -85,B 0,C 180,E1 -9538.138,E2 -9538.138} C_VEL
LIN {X 0,Y 432.725,Z 515.578,A -85,B 0,C 180,E1 -9540,E2 -9540} C_VEL
LIN {X 0,Y 432.598,Z 515.601,A -85,B 0,C 180,E1 -9542.793,E2 -9542.793} C_VEL
LIN {X 0,Y 432.567,Z 515.6,A -85,B 0,C 180,E1 -9546.53,E2 -9546.53} C_VEL
LIN {X 0,Y 432.434,Z 515.62,A -85,B 0,C 180,E1 -9549.353,E2 -9549.353} C_VEL
LIN {X 0,Y 432.422,Z 515.622,A -85,B 0,C 180,E1 -9552.804,E2 -9552.804} C_VEL
LIN {X 0,Y 432.403,Z 515.622,A -85,B 0,C 180,E1 -9556.479,E2 -9556.479} C_VEL
LIN {X 0,Y 432.329,Z 515.63,A -85,B 0,C 180,E1 -9559.96,E2 -9559.96} C_VEL
LIN {X 0,Y 432.31,Z 515.639,A -85,B 0,C 180,E1 -9562.964,E2 -9562.964} C_VEL
LIN {X 0,Y 432.355,Z 515.633,A -85,B 0,C 180,E1 -9566.032,E2 -9566.032} C_VEL
LIN {X 0,Y 432.343,Z 515.635,A -85,B 0,C 180,E1 -9569.187,E2 -9569.187} C_VEL
LIN {X 0,Y 432.406,Z 515.786,A -85,B 0,C 180,E1 -9571.275,E2 -9571.275} C_VEL
LIN {X 0,Y 434.051,Z 524.754,A -85,B 0,C 180,E1 -9573.61,E2 -9573.61} C_VEL
LIN {X 0,Y 437.655,Z 540.315,A -85,B 0,C 180,E1 -9574.057,E2 -9574.057} C_VEL
LIN {X 0,Y 436.589,Z 630.817,A -85,B 0,C 180,E1 -9575.628,E2 -9575.628} C_VEL
LIN {X 0,Y 436.211,Z 644.311,A -85,B 0,C 180,E1 -9576.055,E2 -9576.055} C_VEL
LIN {X 0,Y 435.852,Z 656.451,A -85,B 0,C 180,E1 -9576.627,E2 -9576.627} C_VEL
LIN {X 0,Y 435.243,Z 668.752,A -85,B 0,C 180,E1 -9577.411,E2 -9577.411} C_VEL
LIN {X 0,Y 434.62,Z 680.167,A -85,B 0,C 180,E1 -9578.355,E2 -9578.355} C_VEL
LIN {X 0,Y 433.954,Z 690.866,A -85,B 0,C 180,E1 -9579.469,E2 -9579.469} C_VEL
LIN {X 0,Y 433.244,Z 700.66,A -85,B 0,C 180,E1 -9580.748,E2 -9580.748} C_VEL
LIN {X 0,Y 432.68,Z 708.793,A -85,B 0,C 180,E1 -9582.061,E2 -9582.061} C_VEL
LIN {X 0,Y 432.281,Z 715.359,A -85,B 0,C 180,E1 -9583.367,E2 -9583.367} C_VEL
LIN {X 0,Y 431.891,Z 721.807,A -85,B 0,C 180,E1 -9584.993,E2 -9584.993} C_VEL
LIN {X 0,Y 431.623,Z 725.837,A -85,B 0,C 180,E1 -9586.295,E2 -9586.295} C_VEL
LIN {X 0,Y 431.539,Z 727.905,A -85,B 0,C 180,E1 -9587.126,E2 -9587.126} C_VEL
LIN {X 0,Y 431.336,Z 730.65,A -85,B 0,C 180,E1 -9588.547,E2 -9588.547} C_VEL
LIN {X 0,Y 431.166,Z 732.458,A -85,B 0,C 180,E1 -9590.004,E2 -9590.004} C_VEL
LIN {X 0,Y 431.141,Z 733.322,A -85,B 0,C 180,E1 -9591.726,E2 -9591.726} C_VEL
LIN {X 0,Y 431.16,Z 733.099,A -85,B 0,C 180,E1 -9593.006,E2 -9593.006} C_VEL
LIN {X 0,Y 431.189,Z 731.795,A -85,B 0,C 180,E1 -9594.582,E2 -9594.582} C_VEL
LIN {X 0,Y 431.444,Z 728.92,A -85,B 0,C 180,E1 -9596.37,E2 -9596.37} C_VEL
LIN {X 0,Y 431.594,Z 725.313,A -85,B 0,C 180,E1 -9597.86,E2 -9597.86} C_VEL
LIN {X 0,Y 431.859,Z 721.24,A -85,B 0,C 180,E1 -9599.132,E2 -9599.132} C_VEL
LIN {X 0,Y 432.202,Z 715.625,A -85,B 0,C 180,E1 -9600.536,E2 -9600.536} C_VEL
LIN {X 0,Y 432.579,Z 708.874,A -85,B 0,C 180,E1 -9601.891,E2 -9601.891} C_VEL
LIN {X 0,Y 433.108,Z 700.896,A -85,B 0,C 180,E1 -9603.185,E2 -9603.185} C_VEL
LIN {X 0,Y 433.757,Z 691.327,A -85,B 0,C 180,E1 -9604.445,E2 -9604.445} C_VEL
LIN {X 0,Y 434.358,Z 681.406,A -85,B 0,C 180,E1 -9605.505,E2 -9605.505} C_VEL
LIN {X 0,Y 434.987,Z 669.63,A -85,B 0,C 180,E1 -9606.503,E2 -9606.503} C_VEL
LIN {X 0,Y 435.541,Z 657.863,A -85,B 0,C 180,E1 -9607.279,E2 -9607.279} C_VEL
LIN {X 0,Y 435.972,Z 646.114,A -85,B 0,C 180,E1 -9607.864,E2 -9607.864} C_VEL
LIN {X 0,Y 436.315,Z 633.308,A -85,B 0,C 180,E1 -9608.306,E2 -9608.306} C_VEL
LIN {X 0,Y 436.592,Z 616.09,A -85,B 0,C 180,E1 -9608.647,E2 -9608.647} C_VEL
LIN {X 0,Y 436.614,Z 611.771,A -85,B 0,C 180,E1 -9608.721,E2 -9608.721} C_VEL
LIN {X 0,Y 436.069,Z 605.959,A -85,B 0,C 180,E1 -9608.842,E2 -9608.842} C_VEL
LIN {X 0,Y 430.751,Z 587.257,A -85,B 0,C 180,E1 -9609.375,E2 -9609.375} C_VEL
LIN {X 0,Y 430.168,Z 581.446,A -85,B 0,C 180,E1 -9609.501,E2 -9609.501} C_VEL
LIN {X 0,Y 430.58,Z 540.892,A -85,B 0,C 180,E1 -9610.209,E2 -9610.209} C_VEL
LIN {X 0,Y 426.67,Z 524.102,A -85,B 0,C 180,E1 -9610.68,E2 -9610.68} C_VEL
LIN {X 0,Y 426.568,Z 523.524,A -85,B 0,C 180,E1 -9610.761,E2 -9610.761} C_VEL
LIN {X 0,Y 425.372,Z 516.5,A -85,B 0,C 180,E1 -9612.637,E2 -9612.637} C_VEL
LIN {X 0,Y 425.346,Z 516.498,A -85,B 0,C 180,E1 -9615.65,E2 -9615.65} C_VEL
LIN {X 0,Y 425.349,Z 516.501,A -85,B 0,C 180,E1 -9618.564,E2 -9618.564} C_VEL
LIN {X 0,Y 425.535,Z 516.476,A -85,B 0,C 180,E1 -9622.408,E2 -9622.408} C_VEL
LIN {X 0,Y 425.547,Z 516.474,A -85,B 0,C 180,E1 -9624.313,E2 -9624.313} C_VEL
LIN {X 0,Y 425.573,Z 516.47,A -85,B 0,C 180,E1 -9628.107,E2 -9628.107} C_VEL
LIN {X 0,Y 425.701,Z 516.453,A -85,B 0,C 180,E1 -9630,E2 -9630} C_VEL
LIN {X 0,Y 425.554,Z 516.478,A -85,B 0,C 180,E1 -9632.84,E2 -9632.84} C_VEL
LIN {X 0,Y 425.529,Z 516.479,A -85,B 0,C 180,E1 -9636.639,E2 -9636.639} C_VEL
LIN {X 0,Y 425.398,Z 516.493,A -85,B 0,C 180,E1 -9639.509,E2 -9639.509} C_VEL
LIN {X 0,Y 425.39,Z 516.499,A -85,B 0,C 180,E1 -9642.904,E2 -9642.904} C_VEL
LIN {X 0,Y 425.358,Z 516.499,A -85,B 0,C 180,E1 -9646.605,E2 -9646.605} C_VEL
LIN {X 0,Y 425.325,Z 516.501,A -85,B 0,C 180,E1 -9649.636,E2 -9649.636} C_VEL
LIN {X 0,Y 425.302,Z 516.506,A -85,B 0,C 180,E1 -9653.365,E2 -9653.365} C_VEL
LIN {X 0,Y 425.343,Z 516.504,A -85,B 0,C 180,E1 -9656.844,E2 -9656.844} C_VEL
LIN {X 0,Y 425.314,Z 516.502,A -85,B 0,C 180,E1 -9659.717,E2 -9659.717} C_VEL
LIN {X 0,Y 425.279,Z 516.514,A -85,B 0,C 180,E1 -9663.047,E2 -9663.047} C_VEL
LIN {X 0,Y 425.279,Z 516.506,A -85,B 0,C 180,E1 -9665.929,E2 -9665.929} C_VEL
LIN {X 0,Y 425.308,Z 516.51,A -85,B 0,C 180,E1 -9669.046,E2 -9669.046} C_VEL
LIN {X 0,Y 425.325,Z 516.503,A -85,B 0,C 180,E1 -9672.646,E2 -9672.646} C_VEL
LIN {X 0,Y 425.311,Z 516.502,A -85,B 0,C 180,E1 -9676.051,E2 -9676.051} C_VEL
LIN {X 0,Y 425.302,Z 516.505,A -85,B 0,C 180,E1 -9678.625,E2 -9678.625} C_VEL
LIN {X 0,Y 425.316,Z 516.509,A -85,B 0,C 180,E1 -9681.104,E2 -9681.104} C_VEL
LIN {X 0,Y 425.292,Z 516.507,A -85,B 0,C 180,E1 -9684.664,E2 -9684.664} C_VEL
LIN {X 0,Y 425.257,Z 516.509,A -85,B 0,C 180,E1 -9688.073,E2 -9688.073} C_VEL
LIN {X 0,Y 425.329,Z 516.504,A -85,B 0,C 180,E1 -9691.368,E2 -9691.368} C_VEL
LIN {X 0,Y 425.286,Z 516.506,A -85,B 0,C 180,E1 -9694.555,E2 -9694.555} C_VEL
LIN {X 0,Y 425.278,Z 516.508,A -85,B 0,C 180,E1 -9697.661,E2 -9697.661} C_VEL
LIN {X 0,Y 425.352,Z 516.499,A -85,B 0,C 180,E1 -9700.704,E2 -9700.704} C_VEL
LIN {X 0,Y 425.378,Z 516.495,A -85,B 0,C 180,E1 -9703.688,E2 -9703.688} C_VEL
LIN {X 0,Y 425.421,Z 516.491,A -85,B 0,C 180,E1 -9707.599,E2 -9707.599} C_VEL
LIN {X 0,Y 425.434,Z 516.491,A -85,B 0,C 180,E1 -9711.45,E2 -9711.45} C_VEL
LIN {X 0,Y 425.57,Z 516.47,A -85,B 0,C 180,E1 -9714.314,E2 -9714.314} C_VEL
LIN {X 0,Y 425.567,Z 516.47,A -85,B 0,C 180,E1 -9718.108,E2 -9718.108} C_VEL
LIN {X 0,Y 425.695,Z 516.454,A -85,B 0,C 180,E1 -9720,E2 -9720} C_VEL
LIN {X 0,Y 425.557,Z 516.474,A -85,B 0,C 180,E1 -9722.84,E2 -9722.84} C_VEL
LIN {X 0,Y 425.571,Z 516.472,A -85,B 0,C 180,E1 -9725.687,E2 -9725.687} C_VEL
LIN {X 0,Y 425.434,Z 516.487,A -85,B 0,C 180,E1 -9728.551,E2 -9728.551} C_VEL
LIN {X 0,Y 425.405,Z 516.49,A -85,B 0,C 180,E1 -9732.402,E2 -9732.402} C_VEL
LIN {X 0,Y 425.341,Z 516.505,A -85,B 0,C 180,E1 -9735.33,E2 -9735.33} C_VEL
LIN {X 0,Y 425.325,Z 516.5,A -85,B 0,C 180,E1 -9738.298,E2 -9738.298} C_VEL
LIN {X 0,Y 425.286,Z 516.512,A -85,B 0,C 180,E1 -9741.319,E2 -9741.319} C_VEL
LIN {X 0,Y 425.319,Z 516.502,A -85,B 0,C 180,E1 -9744.66,E2 -9744.66} C_VEL
LIN {X 0,Y 425.344,Z 516.502,A -85,B 0,C 180,E1 -9747.558,E2 -9747.558} C_VEL
LIN {X 0,Y 425.297,Z 516.506,A -85,B 0,C 180,E1 -9750.816,E2 -9750.816} C_VEL
LIN {X 0,Y 425.307,Z 516.502,A -85,B 0,C 180,E1 -9754.289,E2 -9754.289} C_VEL
LIN {X 0,Y 425.282,Z 516.509,A -85,B 0,C 180,E1 -9757.694,E2 -9757.694} C_VEL
LIN {X 0,Y 425.28,Z 516.506,A -85,B 0,C 180,E1 -9760.522,E2 -9760.522} C_VEL
LIN {X 0,Y 425.266,Z 516.509,A -85,B 0,C 180,E1 -9763.956,E2 -9763.956} C_VEL
LIN {X 0,Y 425.33,Z 516.508,A -85,B 0,C 180,E1 -9767.355,E2 -9767.355} C_VEL
LIN {X 0,Y 425.322,Z 516.505,A -85,B 0,C 180,E1 -9771.105,E2 -9771.105} C_VEL
LIN {X 0,Y 425.3,Z 516.504,A -85,B 0,C 180,E1 -9774.665,E2 -9774.665} C_VEL
LIN {X 0,Y 425.265,Z 516.512,A -85,B 0,C 180,E1 -9778.074,E2 -9778.074} C_VEL
LIN {X 0,Y 425.348,Z 516.545,A -85,B 0,C 180,E1 -9781.335,E2 -9781.335} C_VEL
LIN {X 0,Y 428.016,Z 529.213,A -85,B 0,C 180,E1 -9783.923,E2 -9783.923} C_VEL
LIN {X 0,Y 428.74,Z 534.898,A -85,B 0,C 180,E1 -9785.033,E2 -9785.033} C_VEL
LIN {X 0,Y 427.462,Z 554.092,A -85,B 0,C 180,E1 -9788.543,E2 -9788.543} C_VEL
LIN {X 0,Y 426.574,Z 569.425,A -85,B 0,C 180,E1 -9791.31,E2 -9791.31} C_VEL
LIN {X 0,Y 430.324,Z 596.288,A -85,B 0,C 180,E1 -9791.95,E2 -9791.95} C_VEL
LIN {X 0,Y 429.341,Z 678.393,A -85,B 0,C 180,E1 -9793.385,E2 -9793.385} C_VEL
LIN {X 0,Y 428.883,Z 691.514,A -85,B 0,C 180,E1 -9793.795,E2 -9793.795} C_VEL
LIN {X 0,Y 428.381,Z 702.509,A -85,B 0,C 180,E1 -9794.295,E2 -9794.295} C_VEL
LIN {X 0,Y 427.704,Z 714.224,A -85,B 0,C 180,E1 -9795.001,E2 -9795.001} C_VEL
LIN {X 0,Y 427.048,Z 724.966,A -85,B 0,C 180,E1 -9795.834,E2 -9795.834} C_VEL
LIN {X 0,Y 426.381,Z 735.871,A -85,B 0,C 180,E1 -9796.901,E2 -9796.901} C_VEL
LIN {X 0,Y 425.741,Z 745.701,A -85,B 0,C 180,E1 -9798.092,E2 -9798.092} C_VEL
LIN {X 0,Y 425.178,Z 753.756,A -85,B 0,C 180,E1 -9799.283,E2 -9799.283} C_VEL
LIN {X 0,Y 424.739,Z 761.654,A -85,B 0,C 180,E1 -9800.716,E2 -9800.716} C_VEL
LIN {X 0,Y 424.5,Z 767.026,A -85,B 0,C 180,E1 -9801.91,E2 -9801.91} C_VEL
LIN {X 0,Y 424.277,Z 773.225,A -85,B 0,C 180,E1 -9803.66,E2 -9803.66} C_VEL
LIN {X 0,Y 424.217,Z 777.394,A -85,B 0,C 180,E1 -9805.249,E2 -9805.249} C_VEL
LIN {X 0,Y 424.14,Z 779.292,A -85,B 0,C 180,E1 -9806.2,E2 -9806.2} C_VEL
LIN {X 0,Y 424.245,Z 780.732,A -85,B 0,C 180,E1 -9807.151,E2 -9807.151} C_VEL
LIN {X 0,Y 424.207,Z 781.741,A -85,B 0,C 180,E1 -9808.101,E2 -9808.101} C_VEL
LIN {X 0,Y 424.19,Z 782.354,A -85,B 0,C 180,E1 -9809.051,E2 -9809.051} C_VEL
LIN {X 0,Y 424.19,Z 782.573,A -85,B 0,C 180,E1 -9810,E2 -9810} C_VEL
LIN {X 0,Y 424.19,Z 782.354,A -85,B 0,C 180,E1 -9810.949,E2 -9810.949} C_VEL
LIN {X 0,Y 424.207,Z 781.727,A -85,B 0,C 180,E1 -9811.899,E2 -9811.899} C_VEL
LIN {X 0,Y 424.227,Z 780.705,A -85,B 0,C 180,E1 -9812.849,E2 -9812.849} C_VEL
LIN {X 0,Y 424.139,Z 779.271,A -85,B 0,C 180,E1 -9813.8,E2 -9813.8} C_VEL
LIN {X 0,Y 424.234,Z 776.274,A -85,B 0,C 180,E1 -9815.228,E2 -9815.228} C_VEL
LIN {X 0,Y 424.3,Z 772.22,A -85,B 0,C 180,E1 -9816.658,E2 -9816.658} C_VEL
LIN {X 0,Y 424.522,Z 766.004,A -85,B 0,C 180,E1 -9818.329,E2 -9818.329} C_VEL
LIN {X 0,Y 424.871,Z 759.223,A -85,B 0,C 180,E1 -9819.761,E2 -9819.761} C_VEL
LIN {X 0,Y 425.381,Z 750.824,A -85,B 0,C 180,E1 -9821.194,E2 -9821.194} C_VEL
LIN {X 0,Y 425.948,Z 742.222,A -85,B 0,C 180,E1 -9822.386,E2 -9822.386} C_VEL
LIN {X 0,Y 426.59,Z 732.513,A -85,B 0,C 180,E1 -9823.485,E2 -9823.485} C_VEL
LIN {X 0,Y 427.326,Z 721.128,A -85,B 0,C 180,E1 -9824.525,E2 -9824.525} C_VEL
LIN {X 0,Y 428.025,Z 709.646,A -85,B 0,C 180,E1 -9825.353,E2 -9825.353} C_VEL
LIN {X 0,Y 428.658,Z 697.835,A -85,B 0,C 180,E1 -9826,E2 -9826} C_VEL
LIN {X 0,Y 429.249,Z 684.293,A -85,B 0,C 180,E1 -9826.527,E2 -9826.527} C_VEL
LIN {X 0,Y 429.615,Z 672.404,A -85,B 0,C 180,E1 -9826.818,E2 -9826.818} C_VEL
LIN {X 0,Y 430.429,Z 594.81,A -85,B 0,C 180,E1 -9828.169,E2 -9828.169} C_VEL
LIN {X 0,Y 426.568,Z 568.295,A -85,B 0,C 180,E1 -9828.844,E2 -9828.844} C_VEL
LIN {X 0,Y 427.695,Z 549.792,A -85,B 0,C 180,E1 -9832.206,E2 -9832.206} C_VEL
LIN {X 0,Y 428.699,Z 534.824,A -85,B 0,C 180,E1 -9834.969,E2 -9834.969} C_VEL
LIN {X 0,Y 428.259,Z 530.261,A -85,B 0,C 180,E1 -9835.866,E2 -9835.866} C_VEL
LIN {X 0,Y 425.797,Z 518.43,A -85,B 0,C 180,E1 -9838.328,E2 -9838.328} C_VEL
LIN {X 0,Y 425.333,Z 516.504,A -85,B 0,C 180,E1 -9838.771,E2 -9838.771} C_VEL
LIN {X 0,Y 425.266,Z 516.515,A -85,B 0,C 180,E1 -9841.926,E2 -9841.926} C_VEL
LIN {X 0,Y 425.3,Z 516.509,A -85,B 0,C 180,E1 -9845.335,E2 -9845.335} C_VEL
LIN {X 0,Y 425.311,Z 516.507,A -85,B 0,C 180,E1 -9849.045,E2 -9849.045} C_VEL
LIN {X 0,Y 425.33,Z 516.505,A -85,B 0,C 180,E1 -9852.645,E2 -9852.645} C_VEL
LIN {X 0,Y 425.266,Z 516.509,A -85,B 0,C 180,E1 -9856.044,E2 -9856.044} C_VEL
LIN {X 0,Y 425.272,Z 516.512,A -85,B 0,C 180,E1 -9858.621,E2 -9858.621} C_VEL
LIN {X 0,Y 425.309,Z 516.507,A -85,B 0,C 180,E1 -9861.102,E2 -9861.102} C_VEL
LIN {X 0,Y 425.296,Z 516.51,A -85,B 0,C 180,E1 -9864.663,E2 -9864.663} C_VEL
LIN {X 0,Y 425.261,Z 516.51,A -85,B 0,C 180,E1 -9868.072,E2 -9868.072} C_VEL
LIN {X 0,Y 425.332,Z 516.501,A -85,B 0,C 180,E1 -9871.367,E2 -9871.367} C_VEL
LIN {X 0,Y 425.29,Z 516.51,A -85,B 0,C 180,E1 -9874.554,E2 -9874.554} C_VEL
LIN {X 0,Y 425.281,Z 516.507,A -85,B 0,C 180,E1 -9877.66,E2 -9877.66} C_VEL
LIN {X 0,Y 425.355,Z 516.501,A -85,B 0,C 180,E1 -9880.703,E2 -9880.703} C_VEL
LIN {X 0,Y 425.38,Z 516.494,A -85,B 0,C 180,E1 -9883.687,E2 -9883.687} C_VEL
LIN {X 0,Y 425.386,Z 516.496,A -85,B 0,C 180,E1 -9887.095,E2 -9887.095} C_VEL
LIN {X 0,Y 425.394,Z 516.491,A -85,B 0,C 180,E1 -9890.49,E2 -9890.49} C_VEL
LIN {X 0,Y 425.524,Z 516.476,A -85,B 0,C 180,E1 -9893.361,E2 -9893.361} C_VEL
LIN {X 0,Y 425.367,Z 516.5,A -85,B 0,C 180,E1 -9895.261,E2 -9895.261} C_VEL
LIN {X 0,Y 425.567,Z 516.47,A -85,B 0,C 180,E1 -9898.107,E2 -9898.107} C_VEL
LIN {X 0,Y 425.695,Z 516.453,A -85,B 0,C 180,E1 -9900,E2 -9900} C_VEL
LIN {X 0,Y 425.55,Z 516.479,A -85,B 0,C 180,E1 -9902.839,E2 -9902.839} C_VEL
LIN {X 0,Y 425.57,Z 516.471,A -85,B 0,C 180,E1 -9905.686,E2 -9905.686} C_VEL
LIN {X 0,Y 425.433,Z 516.49,A -85,B 0,C 180,E1 -9908.55,E2 -9908.55} C_VEL
LIN {X 0,Y 425.403,Z 516.493,A -85,B 0,C 180,E1 -9912.402,E2 -9912.402} C_VEL
LIN {X 0,Y 425.339,Z 516.504,A -85,B 0,C 180,E1 -9915.329,E2 -9915.329} C_VEL
LIN {X 0,Y 425.323,Z 516.503,A -85,B 0,C 180,E1 -9918.297,E2 -9918.297} C_VEL
LIN {X 0,Y 425.284,Z 516.513,A -85,B 0,C 180,E1 -9921.318,E2 -9921.318} C_VEL
LIN {X 0,Y 425.316,Z 516.51,A -85,B 0,C 180,E1 -9924.659,E2 -9924.659} C_VEL
LIN {X 0,Y 425.341,Z 516.508,A -85,B 0,C 180,E1 -9927.558,E2 -9927.558} C_VEL
LIN {X 0,Y 425.351,Z 516.687,A -85,B 0,C 180,E1 -9931.017,E2 -9931.017} C_VEL
LIN {X 0,Y 426.905,Z 524.991,A -85,B 0,C 180,E1 -9933.266,E2 -9933.266} C_VEL
LIN {X 0,Y 429.743,Z 535.577,A -85,B 0,C 180,E1 -9933.6,E2 -9933.6} C_VEL
LIN {X 0,Y 431.013,Z 542.718,A -85,B 0,C 180,E1 -9933.791,E2 -9933.791} C_VEL
LIN {X 0,Y 429.806,Z 631.542,A -85,B 0,C 180,E1 -9935.362,E2 -9935.362} C_VEL
LIN {X 0,Y 429.423,Z 645.354,A -85,B 0,C 180,E1 -9935.813,E2 -9935.813} C_VEL
LIN {X 0,Y 429.002,Z 657.596,A -85,B 0,C 180,E1 -9936.408,E2 -9936.408} C_VEL
LIN {X 0,Y 428.42,Z 669.14,A -85,B 0,C 180,E1 -9937.162,E2 -9937.162} C_VEL
LIN {X 0,Y 427.738,Z 680.986,A -85,B 0,C 180,E1 -9938.16,E2 -9938.16} C_VEL
LIN {X 0,Y 427.049,Z 690.964,A -85,B 0,C 180,E1 -9939.213,E2 -9939.213} C_VEL
LIN {X 0,Y 426.34,Z 700.733,A -85,B 0,C 180,E1 -9940.502,E2 -9940.502} C_VEL
LIN {X 0,Y 425.729,Z 708.925,A -85,B 0,C 180,E1 -9941.835,E2 -9941.835} C_VEL
LIN {X 0,Y 425.241,Z 716.381,A -85,B 0,C 180,E1 -9943.35,E2 -9943.35} C_VEL
LIN {X 0,Y 424.886,Z 721.551,A -85,B 0,C 180,E1 -9944.664,E2 -9944.664} C_VEL
LIN {X 0,Y 424.541,Z 726.772,A -85,B 0,C 180,E1 -9946.391,E2 -9946.391} C_VEL
LIN {X 0,Y 424.303,Z 730.616,A -85,B 0,C 180,E1 -9948.19,E2 -9948.19} C_VEL
LIN {X 0,Y 424.13,Z 732.685,A -85,B 0,C 180,E1 -9949.742,E2 -9949.742} C_VEL
LIN {X 0,Y 424.07,Z 733.621,A -85,B 0,C 180,E1 -9951.161,E2 -9951.161} C_VEL
LIN {X 0,Y 424.072,Z 733.644,A -85,B 0,C 180,E1 -9952.7,E2 -9952.7} C_VEL
LIN {X 0,Y 424.112,Z 732.275,A -85,B 0,C 180,E1 -9954.551,E2 -9954.551} C_VEL
LIN {X 0,Y 424.269,Z 730.296,A -85,B 0,C 180,E1 -9955.918,E2 -9955.918} C_VEL
LIN {X 0,Y 424.502,Z 726.612,A -85,B 0,C 180,E1 -9957.601,E2 -9957.601} C_VEL
LIN {X 0,Y 424.857,Z 721.301,A -85,B 0,C 180,E1 -9959.336,E2 -9959.336} C_VEL
LIN {X 0,Y 425.206,Z 715.686,A -85,B 0,C 180,E1 -9960.741,E2 -9960.741} C_VEL
LIN {X 0,Y 425.652,Z 708.375,A -85,B 0,C 180,E1 -9962.197,E2 -9962.197} C_VEL
LIN {X 0,Y 426.248,Z 699.836,A -85,B 0,C 180,E1 -9963.566,E2 -9963.566} C_VEL
LIN {X 0,Y 426.811,Z 691.566,A -85,B 0,C 180,E1 -9964.652,E2 -9964.652} C_VEL
LIN {X 0,Y 427.442,Z 681.597,A -85,B 0,C 180,E1 -9965.73,E2 -9965.73} C_VEL
LIN {X 0,Y 428.073,Z 670.746,A -85,B 0,C 180,E1 -9966.667,E2 -9966.667} C_VEL
LIN {X 0,Y 428.658,Z 658.974,A -85,B 0,C 180,E1 -9967.466,E2 -9967.466} C_VEL
LIN {X 0,Y 429.144,Z 645.996,A -85,B 0,C 180,E1 -9968.126,E2 -9968.126} C_VEL
LIN {X 0,Y 429.521,Z 632.944,A -85,B 0,C 180,E1 -9968.572,E2 -9968.572} C_VEL
LIN {X 0,Y 429.772,Z 613.402,A -85,B 0,C 180,E1 -9968.954,E2 -9968.954} C_VEL
LIN {X 0,Y 430.168,Z 581.446,A -85,B 0,C 180,E1 -9969.501,E2 -9969.501} C_VEL
LIN {X 0,Y 429.597,Z 575.639,A -85,B 0,C 180,E1 -9969.627,E2 -9969.627} C_VEL
LIN {X 0,Y 424.377,Z 556.943,A -85,B 0,C 180,E1 -9970.182,E2 -9970.182} C_VEL
LIN {X 0,Y 423.824,Z 551.136,A -85,B 0,C 180,E1 -9970.312,E2 -9970.312} C_VEL
LIN {X 0,Y 423.85,Z 542.123,A -85,B 0,C 180,E1 -9970.476,E2 -9970.476} C_VEL
LIN {X 0,Y 420.254,Z 526.588,A -85,B 0,C 180,E1 -9970.921,E2 -9970.921} C_VEL
LIN {X 0,Y 419.506,Z 524.068,A -85,B 0,C 180,E1 -9971.028,E2 -9971.028} C_VEL
LIN {X 0,Y 418.323,Z 517.379,A -85,B 0,C 180,E1 -9972.838,E2 -9972.838} C_VEL
LIN {X 0,Y 418.311,Z 517.376,A -85,B 0,C 180,E1 -9976.396,E2 -9976.396} C_VEL
LIN {X 0,Y 418.331,Z 517.374,A -85,B 0,C 180,E1 -9979.351,E2 -9979.351} C_VEL
LIN {X 0,Y 418.481,Z 517.354,A -85,B 0,C 180,E1 -9982.279,E2 -9982.279} C_VEL
LIN {X 0,Y 418.506,Z 517.35,A -85,B 0,C 180,E1 -9984.217,E2 -9984.217} C_VEL
LIN {X 0,Y 418.542,Z 517.345,A -85,B 0,C 180,E1 -9988.076,E2 -9988.076} C_VEL
LIN {X 0,Y 418.67,Z 517.329,A -85,B 0,C 180,E1 -9990,E2 -9990} C_VEL
LIN {X 0,Y 418.508,Z 517.357,A -85,B 0,C 180,E1 -9992.888,E2 -9992.888} C_VEL
LIN {X 0,Y 418.491,Z 517.357,A -85,B 0,C 180,E1 -9996.751,E2 -9996.751} C_VEL
LIN {X 0,Y 418.338,Z 517.371,A -85,B 0,C 180,E1 -9999.671,E2 -9999.671} C_VEL
LIN {X 0,Y 418.343,Z 517.377,A -85,B 0,C 180,E1 -10003.001,E2 -10003.001} C_VEL
LIN {X 0,Y 418.309,Z 517.379,A -85,B 0,C 180,E1 -10006.735,E2 -10006.735} C_VEL
LIN {X 0,Y 418.267,Z 517.38,A -85,B 0,C 180,E1 -10009.79,E2 -10009.79} C_VEL
LIN {X 0,Y 418.234,Z 517.388,A -85,B 0,C 180,E1 -10012.736,E2 -10012.736} C_VEL
LIN {X 0,Y 418.266,Z 517.38,A -85,B 0,C 180,E1 -10015.904,E2 -10015.904} C_VEL
LIN {X 0,Y 418.27,Z 517.385,A -85,B 0,C 180,E1 -10019.161,E2 -10019.161} C_VEL
LIN {X 0,Y 418.255,Z 517.386,A -85,B 0,C 180,E1 -10022.844,E2 -10022.844} C_VEL
LIN {X 0,Y 418.243,Z 517.383,A -85,B 0,C 180,E1 -10026.238,E2 -10026.238} C_VEL
LIN {X 0,Y 418.26,Z 517.381,A -85,B 0,C 180,E1 -10029.68,E2 -10029.68} C_VEL
LIN {X 0,Y 418.278,Z 517.379,A -85,B 0,C 180,E1 -10032.329,E2 -10032.329} C_VEL
LIN {X 0,Y 418.267,Z 517.387,A -85,B 0,C 180,E1 -10035.114,E2 -10035.114} C_VEL
LIN {X 0,Y 418.285,Z 517.378,A -85,B 0,C 180,E1 -10037.773,E2 -10037.773} C_VEL
LIN {X 0,Y 418.259,Z 517.383,A -85,B 0,C 180,E1 -10041.56,E2 -10041.56} C_VEL
LIN {X 0,Y 418.251,Z 517.388,A -85,B 0,C 180,E1 -10045.159,E2 -10045.159} C_VEL
LIN {X 0,Y 418.237,Z 517.386,A -85,B 0,C 180,E1 -10047.472,E2 -10047.472} C_VEL
LIN {X 0,Y 418.268,Z 517.384,A -85,B 0,C 180,E1 -10050.893,E2 -10050.893} C_VEL
LIN {X 0,Y 418.262,Z 517.38,A -85,B 0,C 180,E1 -10054.096,E2 -10054.096} C_VEL
LIN {X 0,Y 418.223,Z 517.391,A -85,B 0,C 180,E1 -10057.264,E2 -10057.264} C_VEL
LIN {X 0,Y 418.274,Z 517.379,A -85,B 0,C 180,E1 -10060.364,E2 -10060.364} C_VEL
LIN {X 0,Y 418.307,Z 517.379,A -85,B 0,C 180,E1 -10063.405,E2 -10063.405} C_VEL
LIN {X 0,Y 418.346,Z 517.375,A -85,B 0,C 180,E1 -10066.994,E2 -10066.994} C_VEL
LIN {X 0,Y 418.352,Z 517.369,A -85,B 0,C 180,E1 -10070.329,E2 -10070.329} C_VEL
LIN {X 0,Y 418.487,Z 517.359,A -85,B 0,C 180,E1 -10073.249,E2 -10073.249} C_VEL
LIN {X 0,Y 418.339,Z 517.378,A -85,B 0,C 180,E1 -10075.182,E2 -10075.182} C_VEL
LIN {X 0,Y 418.536,Z 517.346,A -85,B 0,C 180,E1 -10078.076,E2 -10078.076} C_VEL
LIN {X 0,Y 418.665,Z 517.33,A -85,B 0,C 180,E1 -10080,E2 -10080} C_VEL
LIN {X 0,Y 418.51,Z 517.353,A -85,B 0,C 180,E1 -10082.888,E2 -10082.888} C_VEL
LIN {X 0,Y 418.526,Z 517.349,A -85,B 0,C 180,E1 -10085.783,E2 -10085.783} C_VEL
LIN {X 0,Y 418.392,Z 517.366,A -85,B 0,C 180,E1 -10088.696,E2 -10088.696} C_VEL
LIN {X 0,Y 418.309,Z 517.377,A -85,B 0,C 180,E1 -10091.632,E2 -10091.632} C_VEL
LIN {X 0,Y 418.299,Z 517.376,A -85,B 0,C 180,E1 -10094.598,E2 -10094.598} C_VEL
LIN {X 0,Y 418.28,Z 517.381,A -85,B 0,C 180,E1 -10097.605,E2 -10097.605} C_VEL
LIN {X 0,Y 418.243,Z 517.384,A -85,B 0,C 180,E1 -10100.664,E2 -10100.664} C_VEL
LIN {X 0,Y 418.281,Z 517.38,A -85,B 0,C 180,E1 -10103.782,E2 -10103.782} C_VEL
LIN {X 0,Y 418.304,Z 517.38,A -85,B 0,C 180,E1 -10107.071,E2 -10107.071} C_VEL
LIN {X 0,Y 418.258,Z 517.38,A -85,B 0,C 180,E1 -10110.271,E2 -10110.271} C_VEL
LIN {X 0,Y 418.245,Z 517.385,A -85,B 0,C 180,E1 -10113.678,E2 -10113.678} C_VEL
LIN {X 0,Y 418.242,Z 517.389,A -85,B 0,C 180,E1 -10117.225,E2 -10117.225} C_VEL
LIN {X 0,Y 418.252,Z 517.385,A -85,B 0,C 180,E1 -10119.682,E2 -10119.682} C_VEL
LIN {X 0,Y 418.229,Z 517.384,A -85,B 0,C 180,E1 -10122.323,E2 -10122.323} C_VEL
LIN {X 0,Y 418.258,Z 517.385,A -85,B 0,C 180,E1 -10125.113,E2 -10125.113} C_VEL
LIN {X 0,Y 418.29,Z 517.379,A -85,B 0,C 180,E1 -10127.774,E2 -10127.774} C_VEL
LIN {X 0,Y 418.265,Z 517.385,A -85,B 0,C 180,E1 -10131.561,E2 -10131.561} C_VEL
LIN {X 0,Y 418.259,Z 517.385,A -85,B 0,C 180,E1 -10135.16,E2 -10135.16} C_VEL
LIN {X 0,Y 418.246,Z 517.39,A -85,B 0,C 180,E1 -10137.473,E2 -10137.473} C_VEL
LIN {X 0,Y 418.28,Z 517.397,A -85,B 0,C 180,E1 -10141.066,E2 -10141.066} C_VEL
LIN {X 0,Y 421.025,Z 530.261,A -85,B 0,C 180,E1 -10143.747,E2 -10143.747} C_VEL
LIN {X 0,Y 421.802,Z 535.821,A -85,B 0,C 180,E1 -10144.858,E2 -10144.858} C_VEL
LIN {X 0,Y 420.551,Z 553.633,A -85,B 0,C 180,E1 -10148.172,E2 -10148.172} C_VEL
LIN {X 0,Y 419.623,Z 569.03,A -85,B 0,C 180,E1 -10151.002,E2 -10151.002} C_VEL
LIN {X 0,Y 423.519,Z 596.761,A -85,B 0,C 180,E1 -10151.682,E2 -10151.682} C_VEL
LIN {X 0,Y 422.5,Z 678.425,A -85,B 0,C 180,E1 -10153.139,E2 -10153.139} C_VEL
LIN {X 0,Y 422.011,Z 691.4,A -85,B 0,C 180,E1 -10153.554,E2 -10153.554} C_VEL
LIN {X 0,Y 421.471,Z 702.886,A -85,B 0,C 180,E1 -10154.092,E2 -10154.092} C_VEL
LIN {X 0,Y 420.685,Z 715.261,A -85,B 0,C 180,E1 -10154.869,E2 -10154.869} C_VEL
LIN {X 0,Y 419.954,Z 726.943,A -85,B 0,C 180,E1 -10155.834,E2 -10155.834} C_VEL
LIN {X 0,Y 419.273,Z 737.461,A -85,B 0,C 180,E1 -10156.921,E2 -10156.921} C_VEL
LIN {X 0,Y 418.618,Z 746.932,A -85,B 0,C 180,E1 -10158.132,E2 -10158.132} C_VEL
LIN {X 0,Y 417.942,Z 756.068,A -85,B 0,C 180,E1 -10159.586,E2 -10159.586} C_VEL
LIN {X 0,Y 417.552,Z 763.439,A -85,B 0,C 180,E1 -10161.043,E2 -10161.043} C_VEL
LIN {X 0,Y 417.333,Z 768.425,A -85,B 0,C 180,E1 -10162.258,E2 -10162.258} C_VEL
LIN {X 0,Y 417.181,Z 773.197,A -85,B 0,C 180,E1 -10163.692,E2 -10163.692} C_VEL
LIN {X 0,Y 417.147,Z 776.963,A -85,B 0,C 180,E1 -10165.168,E2 -10165.168} C_VEL
LIN {X 0,Y 417.053,Z 778.866,A -85,B 0,C 180,E1 -10166.135,E2 -10166.135} C_VEL
LIN {X 0,Y 417.155,Z 780.313,A -85,B 0,C 180,E1 -10167.103,E2 -10167.103} C_VEL
LIN {X 0,Y 417.132,Z 781.326,A -85,B 0,C 180,E1 -10168.069,E2 -10168.069} C_VEL
LIN {X 0,Y 417.107,Z 781.942,A -85,B 0,C 180,E1 -10169.035,E2 -10169.035} C_VEL
LIN {X 0,Y 417.104,Z 782.164,A -85,B 0,C 180,E1 -10170,E2 -10170} C_VEL
LIN {X 0,Y 417.107,Z 781.948,A -85,B 0,C 180,E1 -10170.965,E2 -10170.965} C_VEL
LIN {X 0,Y 417.131,Z 781.324,A -85,B 0,C 180,E1 -10171.931,E2 -10171.931} C_VEL
LIN {X 0,Y 417.139,Z 780.303,A -85,B 0,C 180,E1 -10172.897,E2 -10172.897} C_VEL
LIN {X 0,Y 417.052,Z 778.872,A -85,B 0,C 180,E1 -10173.865,E2 -10173.865} C_VEL
LIN {X 0,Y 417.146,Z 775.879,A -85,B 0,C 180,E1 -10175.317,E2 -10175.317} C_VEL
LIN {X 0,Y 417.232,Z 771.831,A -85,B 0,C 180,E1 -10176.771,E2 -10176.771} C_VEL
LIN {X 0,Y 417.464,Z 765.623,A -85,B 0,C 180,E1 -10178.471,E2 -10178.471} C_VEL
LIN {X 0,Y 417.843,Z 758.847,A -85,B 0,C 180,E1 -10179.927,E2 -10179.927} C_VEL
LIN {X 0,Y 418.382,Z 750.451,A -85,B 0,C 180,E1 -10181.383,E2 -10181.383} C_VEL
LIN {X 0,Y 418.954,Z 741.858,A -85,B 0,C 180,E1 -10182.596,E2 -10182.596} C_VEL
LIN {X 0,Y 419.66,Z 731.762,A -85,B 0,C 180,E1 -10183.754,E2 -10183.754} C_VEL
LIN {X 0,Y 420.429,Z 720.791,A -85,B 0,C 180,E1 -10184.769,E2 -10184.769} C_VEL
LIN {X 0,Y 421.188,Z 709.334,A -85,B 0,C 180,E1 -10185.608,E2 -10185.608} C_VEL
LIN {X 0,Y 421.84,Z 697.575,A -85,B 0,C 180,E1 -10186.266,E2 -10186.266} C_VEL
LIN {X 0,Y 422.454,Z 684.109,A -85,B 0,C 180,E1 -10186.801,E2 -10186.801} C_VEL
LIN {X 0,Y 422.856,Z 670.913,A -85,B 0,C 180,E1 -10187.127,E2 -10187.127} C_VEL
LIN {X 0,Y 423.761,Z 596.176,A -85,B 0,C 180,E1 -10188.449,E2 -10188.449} C_VEL
LIN {X 0,Y 419.859,Z 569.392,A -85,B 0,C 180,E1 -10189.133,E2 -10189.133} C_VEL
LIN {X 0,Y 419.654,Z 567.857,A -85,B 0,C 180,E1 -10189.184,E2 -10189.184} C_VEL
LIN {X 0,Y 420.744,Z 550.842,A -85,B 0,C 180,E1 -10192.334,E2 -10192.334} C_VEL
LIN {X 0,Y 421.807,Z 535.907,A -85,B 0,C 180,E1 -10195.142,E2 -10195.142} C_VEL
LIN {X 0,Y 421.081,Z 530.467,A -85,B 0,C 180,E1 -10196.249,E2 -10196.249} C_VEL
LIN {X 0,Y 418.764,Z 519.574,A -85,B 0,C 180,E1 -10198.574,E2 -10198.574} C_VEL
LIN {X 0,Y 418.269,Z 517.384,A -85,B 0,C 180,E1 -10199.104,E2 -10199.104} C_VEL
LIN {X 0,Y 418.258,Z 517.387,A -85,B 0,C 180,E1 -10202.843,E2 -10202.843} C_VEL
LIN {X 0,Y 418.248,Z 517.389,A -85,B 0,C 180,E1 -10206.238,E2 -10206.238} C_VEL
LIN {X 0,Y 418.264,Z 517.382,A -85,B 0,C 180,E1 -10209.679,E2 -10209.679} C_VEL
LIN {X 0,Y 418.283,Z 517.383,A -85,B 0,C 180,E1 -10212.329,E2 -10212.329} C_VEL
LIN {X 0,Y 418.252,Z 517.384,A -85,B 0,C 180,E1 -10215.11,E2 -10215.11} C_VEL
LIN {X 0,Y 418.239,Z 517.382,A -85,B 0,C 180,E1 -10217.766,E2 -10217.766} C_VEL
LIN {X 0,Y 418.253,Z 517.385,A -85,B 0,C 180,E1 -10220.618,E2 -10220.618} C_VEL
LIN {X 0,Y 418.242,Z 517.383,A -85,B 0,C 180,E1 -10223.975,E2 -10223.975} C_VEL
LIN {X 0,Y 418.253,Z 517.386,A -85,B 0,C 180,E1 -10227.155,E2 -10227.155} C_VEL
LIN {X 0,Y 418.269,Z 517.386,A -85,B 0,C 180,E1 -10230.838,E2 -10230.838} C_VEL
LIN {X 0,Y 418.265,Z 517.382,A -85,B 0,C 180,E1 -10234.095,E2 -10234.095} C_VEL
LIN {X 0,Y 418.231,Z 517.388,A -85,B 0,C 180,E1 -10237.263,E2 -10237.263} C_VEL
LIN {X 0,Y 418.276,Z 517.379,A -85,B 0,C 180,E1 -10240.363,E2 -10240.363} C_VEL
LIN {X 0,Y 418.309,Z 517.377,A -85,B 0,C 180,E1 -10243.404,E2 -10243.404} C_VEL
LIN {X 0,Y 418.339,Z 517.373,A -85,B 0,C 180,E1 -10246.998,E2 -10246.998} C_VEL
LIN {X 0,Y 418.334,Z 517.37,A -85,B 0,C 180,E1 -10250.328,E2 -10250.328} C_VEL
LIN {X 0,Y 418.487,Z 517.353,A -85,B 0,C 180,E1 -10253.248,E2 -10253.248} C_VEL
LIN {X 0,Y 418.338,Z 517.377,A -85,B 0,C 180,E1 -10255.181,E2 -10255.181} C_VEL
LIN {X 0,Y 418.536,Z 517.346,A -85,B 0,C 180,E1 -10258.075,E2 -10258.075} C_VEL
LIN {X 0,Y 418.665,Z 517.329,A -85,B 0,C 180,E1 -10260,E2 -10260} C_VEL
LIN {X 0,Y 418.504,Z 517.356,A -85,B 0,C 180,E1 -10262.887,E2 -10262.887} C_VEL
LIN {X 0,Y 418.484,Z 517.354,A -85,B 0,C 180,E1 -10266.61,E2 -10266.61} C_VEL
LIN {X 0,Y 418.333,Z 517.375,A -85,B 0,C 180,E1 -10269.671,E2 -10269.671} C_VEL
LIN {X 0,Y 418.337,Z 517.378,A -85,B 0,C 180,E1 -10273.001,E2 -10273.001} C_VEL
LIN {X 0,Y 418.303,Z 517.38,A -85,B 0,C 180,E1 -10276.735,E2 -10276.735} C_VEL
LIN {X 0,Y 418.261,Z 517.384,A -85,B 0,C 180,E1 -10279.79,E2 -10279.79} C_VEL
LIN {X 0,Y 418.229,Z 517.391,A -85,B 0,C 180,E1 -10282.736,E2 -10282.736} C_VEL
LIN {X 0,Y 418.262,Z 517.39,A -85,B 0,C 180,E1 -10285.904,E2 -10285.904} C_VEL
LIN {X 0,Y 418.266,Z 517.388,A -85,B 0,C 180,E1 -10289.161,E2 -10289.161} C_VEL
LIN {X 0,Y 418.27,Z 517.398,A -85,B 0,C 180,E1 -10290.698,E2 -10290.698} C_VEL
